//     PlcTask Inputs/GVL_iXlinker.EtherCAT_Master_EJxxxx.Beckhoff_EJ7xxx.A_0004_EJ7047_0000_0018.ENC_Status_compact.Status/Status_of_input_B <-> ENC Status compact/Status/Status of input B
//     PlcTask Inputs/GVL_iXlinker.EtherCAT_Master_EJxxxx.Beckhoff_EJ7xxx.A_0004_EJ7047_0000_0018.ENC_Status_compact.Status/Status_of_input_C <-> ENC Status compact/Status/Status of input C
//     PlcTask Inputs/GVL_iXlinker.EtherCAT_Master_EJxxxx.Beckhoff_EJ7xxx.A_0004_EJ7047_0000_0018.ENC_Status_compact.Status/Status_of_extern_latch <-> ENC Status compact/Status/Status of extern latch
//     PlcTask Inputs/GVL_iXlinker.EtherCAT_Master_EJxxxx.Beckhoff_EJ7xxx.A_0004_EJ7047_0000_0018.ENC_Status_compact.Status/Sync_error <-> ENC Status compact/Status/Sync error
//     PlcTask Inputs/GVL_iXlinker.EtherCAT_Master_EJxxxx.Beckhoff_EJ7xxx.A_0004_EJ7047_0000_0018.ENC_Status_compact.Status/TxPDO_Toggle <-> ENC Status compact/Status/TxPDO Toggle
//     PlcTask Inputs/GVL_iXlinker.EtherCAT_Master_EJxxxx.Beckhoff_EJ7xxx.A_0004_EJ7047_0000_0018.ENC_Status_compact.Counter_value <-> ENC Status compact/Counter value
//     PlcTask Inputs/GVL_iXlinker.EtherCAT_Master_EJxxxx.Beckhoff_EJ7xxx.A_0004_EJ7047_0000_0018.ENC_Status_compact.Latch_value <-> ENC Status compact/Latch value
//     PlcTask Inputs/GVL_iXlinker.EtherCAT_Master_EJxxxx.Beckhoff_EJ7xxx.A_0004_EJ7047_0000_0018.STM_Status.Status/Ready_to_enable <-> STM Status/Status/Ready to enable
//     PlcTask Inputs/GVL_iXlinker.EtherCAT_Master_EJxxxx.Beckhoff_EJ7xxx.A_0004_EJ7047_0000_0018.STM_Status.Status/Ready <-> STM Status/Status/Ready
//     PlcTask Inputs/GVL_iXlinker.EtherCAT_Master_EJxxxx.Beckhoff_EJ7xxx.A_0004_EJ7047_0000_0018.STM_Status.Status/Warning <-> STM Status/Status/Warning
//     PlcTask Inputs/GVL_iXlinker.EtherCAT_Master_EJxxxx.Beckhoff_EJ7xxx.A_0004_EJ7047_0000_0018.STM_Status.Status/Error <-> STM Status/Status/Error
//     PlcTask Inputs/GVL_iXlinker.EtherCAT_Master_EJxxxx.Beckhoff_EJ7xxx.A_0004_EJ7047_0000_0018.STM_Status.Status/Moving_positive <-> STM Status/Status/Moving positive
//     PlcTask Inputs/GVL_iXlinker.EtherCAT_Master_EJxxxx.Beckhoff_EJ7xxx.A_0004_EJ7047_0000_0018.STM_Status.Status/Moving_negative <-> STM Status/Status/Moving negative
//     PlcTask Inputs/GVL_iXlinker.EtherCAT_Master_EJxxxx.Beckhoff_EJ7xxx.A_0004_EJ7047_0000_0018.STM_Status.Status/Torque_reduced <-> STM Status/Status/Torque reduced
//     PlcTask Inputs/GVL_iXlinker.EtherCAT_Master_EJxxxx.Beckhoff_EJ7xxx.A_0004_EJ7047_0000_0018.STM_Status.Status/Motor_stall <-> STM Status/Status/Motor stall
//     PlcTask Inputs/GVL_iXlinker.EtherCAT_Master_EJxxxx.Beckhoff_EJ7xxx.A_0004_EJ7047_0000_0018.STM_Status.Status/Digital_input_1 <-> STM Status/Status/Digital input 1
//     PlcTask Inputs/GVL_iXlinker.EtherCAT_Master_EJxxxx.Beckhoff_EJ7xxx.A_0004_EJ7047_0000_0018.STM_Status.Status/Digital_input_2 <-> STM Status/Status/Digital input 2
//     PlcTask Inputs/GVL_iXlinker.EtherCAT_Master_EJxxxx.Beckhoff_EJ7xxx.A_0004_EJ7047_0000_0018.STM_Status.Status/Sync_error <-> STM Status/Status/Sync error
//     PlcTask Inputs/GVL_iXlinker.EtherCAT_Master_EJxxxx.Beckhoff_EJ7xxx.A_0004_EJ7047_0000_0018.STM_Status.Status/TxPDO_Toggle <-> STM Status/Status/TxPDO Toggle
//     PlcTask Outputs/GVL_iXlinker.EtherCAT_Master_EJxxxx.Beckhoff_EJ7xxx.A_0004_EJ7047_0000_0018.ENC_Control_compact.Control/Enable_latch_C <-> ENC Control compact/Control/Enable latch C
//     PlcTask Outputs/GVL_iXlinker.EtherCAT_Master_EJxxxx.Beckhoff_EJ7xxx.A_0004_EJ7047_0000_0018.ENC_Control_compact.Control/Enable_latch_extern_on_positive_edge <-> ENC Control compact/Control/Enable latch extern on positive edge
//     PlcTask Outputs/GVL_iXlinker.EtherCAT_Master_EJxxxx.Beckhoff_EJ7xxx.A_0004_EJ7047_0000_0018.ENC_Control_compact.Control/Set_counter <-> ENC Control compact/Control/Set counter
//     PlcTask Outputs/GVL_iXlinker.EtherCAT_Master_EJxxxx.Beckhoff_EJ7xxx.A_0004_EJ7047_0000_0018.ENC_Control_compact.Control/Enable_latch_extern_on_negative_edge <-> ENC Control compact/Control/Enable latch extern on negative edge
//     PlcTask Outputs/GVL_iXlinker.EtherCAT_Master_EJxxxx.Beckhoff_EJ7xxx.A_0004_EJ7047_0000_0018.ENC_Control_compact.Set_counter_value <-> ENC Control compact/Set counter value
//     PlcTask Outputs/GVL_iXlinker.EtherCAT_Master_EJxxxx.Beckhoff_EJ7xxx.A_0004_EJ7047_0000_0018.STM_Control.Control/Enable <-> STM Control/Control/Enable
//     PlcTask Outputs/GVL_iXlinker.EtherCAT_Master_EJxxxx.Beckhoff_EJ7xxx.A_0004_EJ7047_0000_0018.STM_Control.Control/Reset <-> STM Control/Control/Reset
//     PlcTask Outputs/GVL_iXlinker.EtherCAT_Master_EJxxxx.Beckhoff_EJ7xxx.A_0004_EJ7047_0000_0018.STM_Control.Control/Reduce_torque <-> STM Control/Control/Reduce torque
//     PlcTask Outputs/GVL_iXlinker.EtherCAT_Master_EJxxxx.Beckhoff_EJ7xxx.A_0004_EJ7047_0000_0018.STM_Control.Control/Digital_output_1 <-> STM Control/Control/Digital output 1
//     PlcTask Outputs/GVL_iXlinker.EtherCAT_Master_EJxxxx.Beckhoff_EJ7xxx.A_0004_EJ7047_0000_0018.STM_Velocity.Velocity <-> STM Velocity/Velocity
//     PlcTask Inputs/GVL_iXlinker.EtherCAT_Master_EJxxxx.Beckhoff_EJ7xxx.A_0004_EJ7047_0000_0018.WcState.WcState <-> WcState/WcState
//     PlcTask Inputs/GVL_iXlinker.EtherCAT_Master_EJxxxx.Beckhoff_EJ7xxx.A_0004_EJ7047_0000_0018.WcState.InputToggle <-> WcState/InputToggle
//     PlcTask Inputs/GVL_iXlinker.EtherCAT_Master_EJxxxx.Beckhoff_EJ7xxx.A_0004_EJ7047_0000_0018.InfoData.AdsAddr <-> InfoData/AdsAddr
//     PlcTask Inputs/GVL_iXlinker.EtherCAT_Master_EJxxxx.Beckhoff_EJ7xxx.A_0004_EJ7047_0000_0018.InfoData.Chn0 <-> InfoData/Chn0
//     PlcTask Inputs/GVL_iXlinker.EtherCAT_Master_EJxxxx.Beckhoff_EJ7xxx.A_0004_EJ7047_0000_0018.InfoData.Chn1 <-> InfoData/Chn1
//     PlcTask Inputs/GVL_iXlinker.EtherCAT_Master_EJxxxx.Beckhoff_EJ7xxx.A_0004_EJ7047_0000_0018.InfoData.State <-> InfoData/State
//   PLC/PLC Instance <-> EtherCAT Master EJxxxx/Beckhoff EJ7xxx/A_0005(EJ7047-0000-0019)
//     PlcTask Inputs/GVL_iXlinker.EtherCAT_Master_EJxxxx.Beckhoff_EJ7xxx.A_0005_EJ7047_0000_0019.ENC_Status_compact.Status/Latch_C_valid <-> ENC Status compact/Status/Latch C valid
//     PlcTask Inputs/GVL_iXlinker.EtherCAT_Master_EJxxxx.Beckhoff_EJ7xxx.A_0005_EJ7047_0000_0019.ENC_Status_compact.Status/Latch_extern_valid <-> ENC Status compact/Status/Latch extern valid
//     PlcTask Inputs/GVL_iXlinker.EtherCAT_Master_EJxxxx.Beckhoff_EJ7xxx.A_0005_EJ7047_0000_0019.ENC_Status_compact.Status/Set_counter_done <-> ENC Status compact/Status/Set counter done
//     PlcTask Inputs/GVL_iXlinker.EtherCAT_Master_EJxxxx.Beckhoff_EJ7xxx.A_0005_EJ7047_0000_0019.ENC_Status_compact.Status/Counter_underflow <-> ENC Status compact/Status/Counter underflow
//     PlcTask Inputs/GVL_iXlinker.EtherCAT_Master_EJxxxx.Beckhoff_EJ7xxx.A_0005_EJ7047_0000_0019.ENC_Status_compact.Status/Counter_overflow <-> ENC Status compact/Status/Counter overflow
//     PlcTask Inputs/GVL_iXlinker.EtherCAT_Master_EJxxxx.Beckhoff_EJ7xxx.A_0005_EJ7047_0000_0019.ENC_Status_compact.Status/Extrapolation_stall <-> ENC Status compact/Status/Extrapolation stall
//     PlcTask Inputs/GVL_iXlinker.EtherCAT_Master_EJxxxx.Beckhoff_EJ7xxx.A_0005_EJ7047_0000_0019.ENC_Status_compact.Status/Status_of_input_A <-> ENC Status compact/Status/Status of input A
//     PlcTask Inputs/GVL_iXlinker.EtherCAT_Master_EJxxxx.Beckhoff_EJ7xxx.A_0005_EJ7047_0000_0019.ENC_Status_compact.Status/Status_of_input_B <-> ENC Status compact/Status/Status of input B
//     PlcTask Inputs/GVL_iXlinker.EtherCAT_Master_EJxxxx.Beckhoff_EJ7xxx.A_0005_EJ7047_0000_0019.ENC_Status_compact.Status/Status_of_input_C <-> ENC Status compact/Status/Status of input C
//     PlcTask Inputs/GVL_iXlinker.EtherCAT_Master_EJxxxx.Beckhoff_EJ7xxx.A_0005_EJ7047_0000_0019.ENC_Status_compact.Status/Status_of_extern_latch <-> ENC Status compact/Status/Status of extern latch
//     PlcTask Inputs/GVL_iXlinker.EtherCAT_Master_EJxxxx.Beckhoff_EJ7xxx.A_0005_EJ7047_0000_0019.ENC_Status_compact.Status/Sync_error <-> ENC Status compact/Status/Sync error
//     PlcTask Inputs/GVL_iXlinker.EtherCAT_Master_EJxxxx.Beckhoff_EJ7xxx.A_0005_EJ7047_0000_0019.ENC_Status_compact.Status/TxPDO_Toggle <-> ENC Status compact/Status/TxPDO Toggle
//     PlcTask Inputs/GVL_iXlinker.EtherCAT_Master_EJxxxx.Beckhoff_EJ7xxx.A_0005_EJ7047_0000_0019.ENC_Status_compact.Counter_value <-> ENC Status compact/Counter value
//     PlcTask Inputs/GVL_iXlinker.EtherCAT_Master_EJxxxx.Beckhoff_EJ7xxx.A_0005_EJ7047_0000_0019.ENC_Status_compact.Latch_value <-> ENC Status compact/Latch value
//     PlcTask Inputs/GVL_iXlinker.EtherCAT_Master_EJxxxx.Beckhoff_EJ7xxx.A_0005_EJ7047_0000_0019.STM_Status.Status/Ready_to_enable <-> STM Status/Status/Ready to enable
//     PlcTask Inputs/GVL_iXlinker.EtherCAT_Master_EJxxxx.Beckhoff_EJ7xxx.A_0005_EJ7047_0000_0019.STM_Status.Status/Ready <-> STM Status/Status/Ready
//     PlcTask Inputs/GVL_iXlinker.EtherCAT_Master_EJxxxx.Beckhoff_EJ7xxx.A_0005_EJ7047_0000_0019.STM_Status.Status/Warning <-> STM Status/Status/Warning
//     PlcTask Inputs/GVL_iXlinker.EtherCAT_Master_EJxxxx.Beckhoff_EJ7xxx.A_0005_EJ7047_0000_0019.STM_Status.Status/Error <-> STM Status/Status/Error
//     PlcTask Inputs/GVL_iXlinker.EtherCAT_Master_EJxxxx.Beckhoff_EJ7xxx.A_0005_EJ7047_0000_0019.STM_Status.Status/Moving_positive <-> STM Status/Status/Moving positive
//     PlcTask Inputs/GVL_iXlinker.EtherCAT_Master_EJxxxx.Beckhoff_EJ7xxx.A_0005_EJ7047_0000_0019.STM_Status.Status/Moving_negative <-> STM Status/Status/Moving negative
//     PlcTask Inputs/GVL_iXlinker.EtherCAT_Master_EJxxxx.Beckhoff_EJ7xxx.A_0005_EJ7047_0000_0019.STM_Status.Status/Torque_reduced <-> STM Status/Status/Torque reduced
//     PlcTask Inputs/GVL_iXlinker.EtherCAT_Master_EJxxxx.Beckhoff_EJ7xxx.A_0005_EJ7047_0000_0019.STM_Status.Status/Motor_stall <-> STM Status/Status/Motor stall
//     PlcTask Inputs/GVL_iXlinker.EtherCAT_Master_EJxxxx.Beckhoff_EJ7xxx.A_0005_EJ7047_0000_0019.STM_Status.Status/Digital_input_1 <-> STM Status/Status/Digital input 1
//     PlcTask Inputs/GVL_iXlinker.EtherCAT_Master_EJxxxx.Beckhoff_EJ7xxx.A_0005_EJ7047_0000_0019.STM_Status.Status/Digital_input_2 <-> STM Status/Status/Digital input 2
//     PlcTask Inputs/GVL_iXlinker.EtherCAT_Master_EJxxxx.Beckhoff_EJ7xxx.A_0005_EJ7047_0000_0019.STM_Status.Status/Sync_error <-> STM Status/Status/Sync error
//     PlcTask Inputs/GVL_iXlinker.EtherCAT_Master_EJxxxx.Beckhoff_EJ7xxx.A_0005_EJ7047_0000_0019.STM_Status.Status/TxPDO_Toggle <-> STM Status/Status/TxPDO Toggle
//     PlcTask Outputs/GVL_iXlinker.EtherCAT_Master_EJxxxx.Beckhoff_EJ7xxx.A_0005_EJ7047_0000_0019.ENC_Control_compact.Control/Enable_latch_C <-> ENC Control compact/Control/Enable latch C
//     PlcTask Outputs/GVL_iXlinker.EtherCAT_Master_EJxxxx.Beckhoff_EJ7xxx.A_0005_EJ7047_0000_0019.ENC_Control_compact.Control/Enable_latch_extern_on_positive_edge <-> ENC Control compact/Control/Enable latch extern on positive edge
//     PlcTask Outputs/GVL_iXlinker.EtherCAT_Master_EJxxxx.Beckhoff_EJ7xxx.A_0005_EJ7047_0000_0019.ENC_Control_compact.Control/Set_counter <-> ENC Control compact/Control/Set counter
//     PlcTask Outputs/GVL_iXlinker.EtherCAT_Master_EJxxxx.Beckhoff_EJ7xxx.A_0005_EJ7047_0000_0019.ENC_Control_compact.Control/Enable_latch_extern_on_negative_edge <-> ENC Control compact/Control/Enable latch extern on negative edge
//     PlcTask Outputs/GVL_iXlinker.EtherCAT_Master_EJxxxx.Beckhoff_EJ7xxx.A_0005_EJ7047_0000_0019.ENC_Control_compact.Set_counter_value <-> ENC Control compact/Set counter value
//     PlcTask Outputs/GVL_iXlinker.EtherCAT_Master_EJxxxx.Beckhoff_EJ7xxx.A_0005_EJ7047_0000_0019.STM_Control.Control/Enable <-> STM Control/Control/Enable
//     PlcTask Outputs/GVL_iXlinker.EtherCAT_Master_EJxxxx.Beckhoff_EJ7xxx.A_0005_EJ7047_0000_0019.STM_Control.Control/Reset <-> STM Control/Control/Reset
//     PlcTask Outputs/GVL_iXlinker.EtherCAT_Master_EJxxxx.Beckhoff_EJ7xxx.A_0005_EJ7047_0000_0019.STM_Control.Control/Reduce_torque <-> STM Control/Control/Reduce torque
//     PlcTask Outputs/GVL_iXlinker.EtherCAT_Master_EJxxxx.Beckhoff_EJ7xxx.A_0005_EJ7047_0000_0019.STM_Control.Control/Digital_output_1 <-> STM Control/Control/Digital output 1
//     PlcTask Outputs/GVL_iXlinker.EtherCAT_Master_EJxxxx.Beckhoff_EJ7xxx.A_0005_EJ7047_0000_0019.STM_Velocity.Velocity <-> STM Velocity/Velocity
//     PlcTask Inputs/GVL_iXlinker.EtherCAT_Master_EJxxxx.Beckhoff_EJ7xxx.A_0005_EJ7047_0000_0019.WcState.WcState <-> WcState/WcState
//     PlcTask Inputs/GVL_iXlinker.EtherCAT_Master_EJxxxx.Beckhoff_EJ7xxx.A_0005_EJ7047_0000_0019.WcState.InputToggle <-> WcState/InputToggle
//     PlcTask Inputs/GVL_iXlinker.EtherCAT_Master_EJxxxx.Beckhoff_EJ7xxx.A_0005_EJ7047_0000_0019.InfoData.AdsAddr <-> InfoData/AdsAddr
//     PlcTask Inputs/GVL_iXlinker.EtherCAT_Master_EJxxxx.Beckhoff_EJ7xxx.A_0005_EJ7047_0000_0019.InfoData.Chn0 <-> InfoData/Chn0
//     PlcTask Inputs/GVL_iXlinker.EtherCAT_Master_EJxxxx.Beckhoff_EJ7xxx.A_0005_EJ7047_0000_0019.InfoData.Chn1 <-> InfoData/Chn1
//     PlcTask Inputs/GVL_iXlinker.EtherCAT_Master_EJxxxx.Beckhoff_EJ7xxx.A_0005_EJ7047_0000_0019.InfoData.State <-> InfoData/State
//   PLC/PLC Instance <-> EtherCAT Master EJxxxx/Beckhoff EJ7xxx/A_0006(EJ7047-0000-0020)
//     PlcTask Inputs/GVL_iXlinker.EtherCAT_Master_EJxxxx.Beckhoff_EJ7xxx.A_0006_EJ7047_0000_0020.ENC_Status_compact.Status/Latch_C_valid <-> ENC Status compact/Status/Latch C valid
//     PlcTask Inputs/GVL_iXlinker.EtherCAT_Master_EJxxxx.Beckhoff_EJ7xxx.A_0006_EJ7047_0000_0020.ENC_Status_compact.Status/Latch_extern_valid <-> ENC Status compact/Status/Latch extern valid
//     PlcTask Inputs/GVL_iXlinker.EtherCAT_Master_EJxxxx.Beckhoff_EJ7xxx.A_0006_EJ7047_0000_0020.ENC_Status_compact.Status/Set_counter_done <-> ENC Status compact/Status/Set counter done
//     PlcTask Inputs/GVL_iXlinker.EtherCAT_Master_EJxxxx.Beckhoff_EJ7xxx.A_0006_EJ7047_0000_0020.ENC_Status_compact.Status/Counter_underflow <-> ENC Status compact/Status/Counter underflow
//     PlcTask Inputs/GVL_iXlinker.EtherCAT_Master_EJxxxx.Beckhoff_EJ7xxx.A_0006_EJ7047_0000_0020.ENC_Status_compact.Status/Counter_overflow <-> ENC Status compact/Status/Counter overflow
//     PlcTask Inputs/GVL_iXlinker.EtherCAT_Master_EJxxxx.Beckhoff_EJ7xxx.A_0006_EJ7047_0000_0020.ENC_Status_compact.Status/Extrapolation_stall <-> ENC Status compact/Status/Extrapolation stall
//     PlcTask Inputs/GVL_iXlinker.EtherCAT_Master_EJxxxx.Beckhoff_EJ7xxx.A_0006_EJ7047_0000_0020.ENC_Status_compact.Status/Status_of_input_A <-> ENC Status compact/Status/Status of input A
//     PlcTask Inputs/GVL_iXlinker.EtherCAT_Master_EJxxxx.Beckhoff_EJ7xxx.A_0006_EJ7047_0000_0020.ENC_Status_compact.Status/Status_of_input_B <-> ENC Status compact/Status/Status of input B
//     PlcTask Inputs/GVL_iXlinker.EtherCAT_Master_EJxxxx.Beckhoff_EJ7xxx.A_0006_EJ7047_0000_0020.ENC_Status_compact.Status/Status_of_input_C <-> ENC Status compact/Status/Status of input C
//     PlcTask Inputs/GVL_iXlinker.EtherCAT_Master_EJxxxx.Beckhoff_EJ7xxx.A_0006_EJ7047_0000_0020.ENC_Status_compact.Status/Status_of_extern_latch <-> ENC Status compact/Status/Status of extern latch
//     PlcTask Inputs/GVL_iXlinker.EtherCAT_Master_EJxxxx.Beckhoff_EJ7xxx.A_0006_EJ7047_0000_0020.ENC_Status_compact.Status/Sync_error <-> ENC Status compact/Status/Sync error
//     PlcTask Inputs/GVL_iXlinker.EtherCAT_Master_EJxxxx.Beckhoff_EJ7xxx.A_0006_EJ7047_0000_0020.ENC_Status_compact.Status/TxPDO_Toggle <-> ENC Status compact/Status/TxPDO Toggle
//     PlcTask Inputs/GVL_iXlinker.EtherCAT_Master_EJxxxx.Beckhoff_EJ7xxx.A_0006_EJ7047_0000_0020.ENC_Status_compact.Counter_value <-> ENC Status compact/Counter value
//     PlcTask Inputs/GVL_iXlinker.EtherCAT_Master_EJxxxx.Beckhoff_EJ7xxx.A_0006_EJ7047_0000_0020.ENC_Status_compact.Latch_value <-> ENC Status compact/Latch value
//     PlcTask Inputs/GVL_iXlinker.EtherCAT_Master_EJxxxx.Beckhoff_EJ7xxx.A_0006_EJ7047_0000_0020.STM_Status.Status/Ready_to_enable <-> STM Status/Status/Ready to enable
//     PlcTask Inputs/GVL_iXlinker.EtherCAT_Master_EJxxxx.Beckhoff_EJ7xxx.A_0006_EJ7047_0000_0020.STM_Status.Status/Ready <-> STM Status/Status/Ready
//     PlcTask Inputs/GVL_iXlinker.EtherCAT_Master_EJxxxx.Beckhoff_EJ7xxx.A_0006_EJ7047_0000_0020.STM_Status.Status/Warning <-> STM Status/Status/Warning
//     PlcTask Inputs/GVL_iXlinker.EtherCAT_Master_EJxxxx.Beckhoff_EJ7xxx.A_0006_EJ7047_0000_0020.STM_Status.Status/Error <-> STM Status/Status/Error
//     PlcTask Inputs/GVL_iXlinker.EtherCAT_Master_EJxxxx.Beckhoff_EJ7xxx.A_0006_EJ7047_0000_0020.STM_Status.Status/Moving_positive <-> STM Status/Status/Moving positive
//     PlcTask Inputs/GVL_iXlinker.EtherCAT_Master_EJxxxx.Beckhoff_EJ7xxx.A_0006_EJ7047_0000_0020.STM_Status.Status/Moving_negative <-> STM Status/Status/Moving negative
//     PlcTask Inputs/GVL_iXlinker.EtherCAT_Master_EJxxxx.Beckhoff_EJ7xxx.A_0006_EJ7047_0000_0020.STM_Status.Status/Torque_reduced <-> STM Status/Status/Torque reduced
//     PlcTask Inputs/GVL_iXlinker.EtherCAT_Master_EJxxxx.Beckhoff_EJ7xxx.A_0006_EJ7047_0000_0020.STM_Status.Status/Motor_stall <-> STM Status/Status/Motor stall
//     PlcTask Inputs/GVL_iXlinker.EtherCAT_Master_EJxxxx.Beckhoff_EJ7xxx.A_0006_EJ7047_0000_0020.STM_Status.Status/Digital_input_1 <-> STM Status/Status/Digital input 1
//     PlcTask Inputs/GVL_iXlinker.EtherCAT_Master_EJxxxx.Beckhoff_EJ7xxx.A_0006_EJ7047_0000_0020.STM_Status.Status/Digital_input_2 <-> STM Status/Status/Digital input 2
//     PlcTask Inputs/GVL_iXlinker.EtherCAT_Master_EJxxxx.Beckhoff_EJ7xxx.A_0006_EJ7047_0000_0020.STM_Status.Status/Sync_error <-> STM Status/Status/Sync error
//     PlcTask Inputs/GVL_iXlinker.EtherCAT_Master_EJxxxx.Beckhoff_EJ7xxx.A_0006_EJ7047_0000_0020.STM_Status.Status/TxPDO_Toggle <-> STM Status/Status/TxPDO Toggle
//     PlcTask Outputs/GVL_iXlinker.EtherCAT_Master_EJxxxx.Beckhoff_EJ7xxx.A_0006_EJ7047_0000_0020.ENC_Control_compact.Control/Enable_latch_C <-> ENC Control compact/Control/Enable latch C
//     PlcTask Outputs/GVL_iXlinker.EtherCAT_Master_EJxxxx.Beckhoff_EJ7xxx.A_0006_EJ7047_0000_0020.ENC_Control_compact.Control/Enable_latch_extern_on_positive_edge <-> ENC Control compact/Control/Enable latch extern on positive edge
//     PlcTask Outputs/GVL_iXlinker.EtherCAT_Master_EJxxxx.Beckhoff_EJ7xxx.A_0006_EJ7047_0000_0020.ENC_Control_compact.Control/Set_counter <-> ENC Control compact/Control/Set counter
//     PlcTask Outputs/GVL_iXlinker.EtherCAT_Master_EJxxxx.Beckhoff_EJ7xxx.A_0006_EJ7047_0000_0020.ENC_Control_compact.Control/Enable_latch_extern_on_negative_edge <-> ENC Control compact/Control/Enable latch extern on negative edge
//     PlcTask Outputs/GVL_iXlinker.EtherCAT_Master_EJxxxx.Beckhoff_EJ7xxx.A_0006_EJ7047_0000_0020.ENC_Control_compact.Set_counter_value <-> ENC Control compact/Set counter value
//     PlcTask Outputs/GVL_iXlinker.EtherCAT_Master_EJxxxx.Beckhoff_EJ7xxx.A_0006_EJ7047_0000_0020.STM_Control.Control/Enable <-> STM Control/Control/Enable
//     PlcTask Outputs/GVL_iXlinker.EtherCAT_Master_EJxxxx.Beckhoff_EJ7xxx.A_0006_EJ7047_0000_0020.STM_Control.Control/Reset <-> STM Control/Control/Reset
//     PlcTask Outputs/GVL_iXlinker.EtherCAT_Master_EJxxxx.Beckhoff_EJ7xxx.A_0006_EJ7047_0000_0020.STM_Control.Control/Reduce_torque <-> STM Control/Control/Reduce torque
//     PlcTask Outputs/GVL_iXlinker.EtherCAT_Master_EJxxxx.Beckhoff_EJ7xxx.A_0006_EJ7047_0000_0020.STM_Control.Control/Digital_output_1 <-> STM Control/Control/Digital output 1
//     PlcTask Outputs/GVL_iXlinker.EtherCAT_Master_EJxxxx.Beckhoff_EJ7xxx.A_0006_EJ7047_0000_0020.STM_Velocity.Velocity <-> STM Velocity/Velocity
//     PlcTask Inputs/GVL_iXlinker.EtherCAT_Master_EJxxxx.Beckhoff_EJ7xxx.A_0006_EJ7047_0000_0020.WcState.WcState <-> WcState/WcState
//     PlcTask Inputs/GVL_iXlinker.EtherCAT_Master_EJxxxx.Beckhoff_EJ7xxx.A_0006_EJ7047_0000_0020.WcState.InputToggle <-> WcState/InputToggle
//     PlcTask Inputs/GVL_iXlinker.EtherCAT_Master_EJxxxx.Beckhoff_EJ7xxx.A_0006_EJ7047_0000_0020.InfoData.AdsAddr <-> InfoData/AdsAddr
//     PlcTask Inputs/GVL_iXlinker.EtherCAT_Master_EJxxxx.Beckhoff_EJ7xxx.A_0006_EJ7047_0000_0020.InfoData.Chn0 <-> InfoData/Chn0
//     PlcTask Inputs/GVL_iXlinker.EtherCAT_Master_EJxxxx.Beckhoff_EJ7xxx.A_0006_EJ7047_0000_0020.InfoData.Chn1 <-> InfoData/Chn1
//     PlcTask Inputs/GVL_iXlinker.EtherCAT_Master_EJxxxx.Beckhoff_EJ7xxx.A_0006_EJ7047_0000_0020.InfoData.State <-> InfoData/State
//   PLC/PLC Instance <-> EtherCAT Master EJxxxx/Beckhoff EJ7xxx/A_0007(EJ7342-0000-0019)
//     PlcTask Inputs/GVL_iXlinker.EtherCAT_Master_EJxxxx.Beckhoff_EJ7xxx.A_0007_EJ7342_0000_0019.ENC_Status_compact_Channel_1.Status/Latch_extern_valid <-> ENC Status compact Channel 1/Status/Latch extern valid
//     PlcTask Inputs/GVL_iXlinker.EtherCAT_Master_EJxxxx.Beckhoff_EJ7xxx.A_0007_EJ7342_0000_0019.ENC_Status_compact_Channel_2.Status/Latch_extern_valid <-> ENC Status compact Channel 2/Status/Latch extern valid
//     PlcTask Inputs/GVL_iXlinker.EtherCAT_Master_EJxxxx.Beckhoff_EJ7xxx.A_0007_EJ7342_0000_0019.ENC_Status_compact_Channel_1.Status/Set_counter_done <-> ENC Status compact Channel 1/Status/Set counter done
//     PlcTask Inputs/GVL_iXlinker.EtherCAT_Master_EJxxxx.Beckhoff_EJ7xxx.A_0007_EJ7342_0000_0019.ENC_Status_compact_Channel_2.Status/Set_counter_done <-> ENC Status compact Channel 2/Status/Set counter done
//     PlcTask Inputs/GVL_iXlinker.EtherCAT_Master_EJxxxx.Beckhoff_EJ7xxx.A_0007_EJ7342_0000_0019.ENC_Status_compact_Channel_1.Status/Counter_underflow <-> ENC Status compact Channel 1/Status/Counter underflow
//     PlcTask Inputs/GVL_iXlinker.EtherCAT_Master_EJxxxx.Beckhoff_EJ7xxx.A_0007_EJ7342_0000_0019.ENC_Status_compact_Channel_2.Status/Counter_underflow <-> ENC Status compact Channel 2/Status/Counter underflow
//     PlcTask Inputs/GVL_iXlinker.EtherCAT_Master_EJxxxx.Beckhoff_EJ7xxx.A_0007_EJ7342_0000_0019.ENC_Status_compact_Channel_1.Status/Counter_overflow <-> ENC Status compact Channel 1/Status/Counter overflow
//     PlcTask Inputs/GVL_iXlinker.EtherCAT_Master_EJxxxx.Beckhoff_EJ7xxx.A_0007_EJ7342_0000_0019.ENC_Status_compact_Channel_2.Status/Counter_overflow <-> ENC Status compact Channel 2/Status/Counter overflow
//     PlcTask Inputs/GVL_iXlinker.EtherCAT_Master_EJxxxx.Beckhoff_EJ7xxx.A_0007_EJ7342_0000_0019.ENC_Status_compact_Channel_1.Status/Extrapolation_stall <-> ENC Status compact Channel 1/Status/Extrapolation stall
//     PlcTask Inputs/GVL_iXlinker.EtherCAT_Master_EJxxxx.Beckhoff_EJ7xxx.A_0007_EJ7342_0000_0019.ENC_Status_compact_Channel_2.Status/Extrapolation_stall <-> ENC Status compact Channel 2/Status/Extrapolation stall
//     PlcTask Inputs/GVL_iXlinker.EtherCAT_Master_EJxxxx.Beckhoff_EJ7xxx.A_0007_EJ7342_0000_0019.ENC_Status_compact_Channel_1.Status/Status_of_input_A <-> ENC Status compact Channel 1/Status/Status of input A
//     PlcTask Inputs/GVL_iXlinker.EtherCAT_Master_EJxxxx.Beckhoff_EJ7xxx.A_0007_EJ7342_0000_0019.ENC_Status_compact_Channel_2.Status/Status_of_input_A <-> ENC Status compact Channel 2/Status/Status of input A
//     PlcTask Inputs/GVL_iXlinker.EtherCAT_Master_EJxxxx.Beckhoff_EJ7xxx.A_0007_EJ7342_0000_0019.ENC_Status_compact_Channel_1.Status/Status_of_input_B <-> ENC Status compact Channel 1/Status/Status of input B
//     PlcTask Inputs/GVL_iXlinker.EtherCAT_Master_EJxxxx.Beckhoff_EJ7xxx.A_0007_EJ7342_0000_0019.ENC_Status_compact_Channel_2.Status/Status_of_input_B <-> ENC Status compact Channel 2/Status/Status of input B
//     PlcTask Inputs/GVL_iXlinker.EtherCAT_Master_EJxxxx.Beckhoff_EJ7xxx.A_0007_EJ7342_0000_0019.ENC_Status_compact_Channel_1.Status/Status_of_extern_latch <-> ENC Status compact Channel 1/Status/Status of extern latch
//     PlcTask Inputs/GVL_iXlinker.EtherCAT_Master_EJxxxx.Beckhoff_EJ7xxx.A_0007_EJ7342_0000_0019.ENC_Status_compact_Channel_2.Status/Status_of_extern_latch <-> ENC Status compact Channel 2/Status/Status of extern latch
//     PlcTask Inputs/GVL_iXlinker.EtherCAT_Master_EJxxxx.Beckhoff_EJ7xxx.A_0007_EJ7342_0000_0019.ENC_Status_compact_Channel_1.Status/Sync_error <-> ENC Status compact Channel 1/Status/Sync error
//     PlcTask Inputs/GVL_iXlinker.EtherCAT_Master_EJxxxx.Beckhoff_EJ7xxx.A_0007_EJ7342_0000_0019.ENC_Status_compact_Channel_2.Status/Sync_error <-> ENC Status compact Channel 2/Status/Sync error
//     PlcTask Inputs/GVL_iXlinker.EtherCAT_Master_EJxxxx.Beckhoff_EJ7xxx.A_0007_EJ7342_0000_0019.ENC_Status_compact_Channel_1.Status/TxPDO_Toggle <-> ENC Status compact Channel 1/Status/TxPDO Toggle
//     PlcTask Inputs/GVL_iXlinker.EtherCAT_Master_EJxxxx.Beckhoff_EJ7xxx.A_0007_EJ7342_0000_0019.ENC_Status_compact_Channel_2.Status/TxPDO_Toggle <-> ENC Status compact Channel 2/Status/TxPDO Toggle
//     PlcTask Inputs/GVL_iXlinker.EtherCAT_Master_EJxxxx.Beckhoff_EJ7xxx.A_0007_EJ7342_0000_0019.ENC_Status_compact_Channel_1.Counter_value <-> ENC Status compact Channel 1/Counter value
//     PlcTask Inputs/GVL_iXlinker.EtherCAT_Master_EJxxxx.Beckhoff_EJ7xxx.A_0007_EJ7342_0000_0019.ENC_Status_compact_Channel_2.Counter_value <-> ENC Status compact Channel 2/Counter value
//     PlcTask Inputs/GVL_iXlinker.EtherCAT_Master_EJxxxx.Beckhoff_EJ7xxx.A_0007_EJ7342_0000_0019.ENC_Status_compact_Channel_1.Latch_value <-> ENC Status compact Channel 1/Latch value
//     PlcTask Inputs/GVL_iXlinker.EtherCAT_Master_EJxxxx.Beckhoff_EJ7xxx.A_0007_EJ7342_0000_0019.ENC_Status_compact_Channel_2.Latch_value <-> ENC Status compact Channel 2/Latch value
//     PlcTask Inputs/GVL_iXlinker.EtherCAT_Master_EJxxxx.Beckhoff_EJ7xxx.A_0007_EJ7342_0000_0019.DCM_Status_Channel_1.Status/Ready_to_enable <-> DCM Status Channel 1/Status/Ready to enable
//     PlcTask Inputs/GVL_iXlinker.EtherCAT_Master_EJxxxx.Beckhoff_EJ7xxx.A_0007_EJ7342_0000_0019.DCM_Status_Channel_2.Status/Ready_to_enable <-> DCM Status Channel 2/Status/Ready to enable
//     PlcTask Inputs/GVL_iXlinker.EtherCAT_Master_EJxxxx.Beckhoff_EJ7xxx.A_0007_EJ7342_0000_0019.DCM_Status_Channel_1.Status/Ready <-> DCM Status Channel 1/Status/Ready
//     PlcTask Inputs/GVL_iXlinker.EtherCAT_Master_EJxxxx.Beckhoff_EJ7xxx.A_0007_EJ7342_0000_0019.DCM_Status_Channel_2.Status/Ready <-> DCM Status Channel 2/Status/Ready
//     PlcTask Inputs/GVL_iXlinker.EtherCAT_Master_EJxxxx.Beckhoff_EJ7xxx.A_0007_EJ7342_0000_0019.DCM_Status_Channel_1.Status/Warning <-> DCM Status Channel 1/Status/Warning
//     PlcTask Inputs/GVL_iXlinker.EtherCAT_Master_EJxxxx.Beckhoff_EJ7xxx.A_0007_EJ7342_0000_0019.DCM_Status_Channel_2.Status/Warning <-> DCM Status Channel 2/Status/Warning
//     PlcTask Inputs/GVL_iXlinker.EtherCAT_Master_EJxxxx.Beckhoff_EJ7xxx.A_0007_EJ7342_0000_0019.DCM_Status_Channel_1.Status/Error <-> DCM Status Channel 1/Status/Error
//     PlcTask Inputs/GVL_iXlinker.EtherCAT_Master_EJxxxx.Beckhoff_EJ7xxx.A_0007_EJ7342_0000_0019.DCM_Status_Channel_2.Status/Error <-> DCM Status Channel 2/Status/Error
//     PlcTask Inputs/GVL_iXlinker.EtherCAT_Master_EJxxxx.Beckhoff_EJ7xxx.A_0007_EJ7342_0000_0019.DCM_Status_Channel_1.Status/Moving_positive <-> DCM Status Channel 1/Status/Moving positive
//     PlcTask Inputs/GVL_iXlinker.EtherCAT_Master_EJxxxx.Beckhoff_EJ7xxx.A_0007_EJ7342_0000_0019.DCM_Status_Channel_2.Status/Moving_positive <-> DCM Status Channel 2/Status/Moving positive
//     PlcTask Inputs/GVL_iXlinker.EtherCAT_Master_EJxxxx.Beckhoff_EJ7xxx.A_0007_EJ7342_0000_0019.DCM_Status_Channel_1.Status/Moving_negative <-> DCM Status Channel 1/Status/Moving negative
//     PlcTask Inputs/GVL_iXlinker.EtherCAT_Master_EJxxxx.Beckhoff_EJ7xxx.A_0007_EJ7342_0000_0019.DCM_Status_Channel_2.Status/Moving_negative <-> DCM Status Channel 2/Status/Moving negative
//     PlcTask Inputs/GVL_iXlinker.EtherCAT_Master_EJxxxx.Beckhoff_EJ7xxx.A_0007_EJ7342_0000_0019.DCM_Status_Channel_1.Status/Torque_reduced <-> DCM Status Channel 1/Status/Torque reduced
//     PlcTask Inputs/GVL_iXlinker.EtherCAT_Master_EJxxxx.Beckhoff_EJ7xxx.A_0007_EJ7342_0000_0019.DCM_Status_Channel_2.Status/Torque_reduced <-> DCM Status Channel 2/Status/Torque reduced
//     PlcTask Inputs/GVL_iXlinker.EtherCAT_Master_EJxxxx.Beckhoff_EJ7xxx.A_0007_EJ7342_0000_0019.DCM_Status_Channel_1.Status/Digital_input_1 <-> DCM Status Channel 1/Status/Digital input 1
//     PlcTask Inputs/GVL_iXlinker.EtherCAT_Master_EJxxxx.Beckhoff_EJ7xxx.A_0007_EJ7342_0000_0019.DCM_Status_Channel_1.Status/Digital_input_2 <-> DCM Status Channel 1/Status/Digital input 2
//     PlcTask Inputs/GVL_iXlinker.EtherCAT_Master_EJxxxx.Beckhoff_EJ7xxx.A_0007_EJ7342_0000_0019.DCM_Status_Channel_2.Status/Digital_input_1 <-> DCM Status Channel 2/Status/Digital input 1
//     PlcTask Inputs/GVL_iXlinker.EtherCAT_Master_EJxxxx.Beckhoff_EJ7xxx.A_0007_EJ7342_0000_0019.DCM_Status_Channel_2.Status/Digital_input_2 <-> DCM Status Channel 2/Status/Digital input 2
//     PlcTask Inputs/GVL_iXlinker.EtherCAT_Master_EJxxxx.Beckhoff_EJ7xxx.A_0007_EJ7342_0000_0019.DCM_Status_Channel_1.Status/Sync_error <-> DCM Status Channel 1/Status/Sync error
//     PlcTask Inputs/GVL_iXlinker.EtherCAT_Master_EJxxxx.Beckhoff_EJ7xxx.A_0007_EJ7342_0000_0019.DCM_Status_Channel_2.Status/Sync_error <-> DCM Status Channel 2/Status/Sync error
//     PlcTask Inputs/GVL_iXlinker.EtherCAT_Master_EJxxxx.Beckhoff_EJ7xxx.A_0007_EJ7342_0000_0019.DCM_Status_Channel_1.Status/TxPDO_Toggle <-> DCM Status Channel 1/Status/TxPDO Toggle
//     PlcTask Inputs/GVL_iXlinker.EtherCAT_Master_EJxxxx.Beckhoff_EJ7xxx.A_0007_EJ7342_0000_0019.DCM_Status_Channel_2.Status/TxPDO_Toggle <-> DCM Status Channel 2/Status/TxPDO Toggle
//     PlcTask Outputs/GVL_iXlinker.EtherCAT_Master_EJxxxx.Beckhoff_EJ7xxx.A_0007_EJ7342_0000_0019.ENC_Control_compact_Channel_1.Control/Enable_latch_extern_on_positive_edge <-> ENC Control compact Channel 1/Control/Enable latch extern on positive edge
//     PlcTask Outputs/GVL_iXlinker.EtherCAT_Master_EJxxxx.Beckhoff_EJ7xxx.A_0007_EJ7342_0000_0019.ENC_Control_compact_Channel_2.Control/Enable_latch_extern_on_positive_edge <-> ENC Control compact Channel 2/Control/Enable latch extern on positive edge
//     PlcTask Outputs/GVL_iXlinker.EtherCAT_Master_EJxxxx.Beckhoff_EJ7xxx.A_0007_EJ7342_0000_0019.ENC_Control_compact_Channel_1.Control/Set_counter <-> ENC Control compact Channel 1/Control/Set counter
//     PlcTask Outputs/GVL_iXlinker.EtherCAT_Master_EJxxxx.Beckhoff_EJ7xxx.A_0007_EJ7342_0000_0019.ENC_Control_compact_Channel_2.Control/Set_counter <-> ENC Control compact Channel 2/Control/Set counter
//     PlcTask Outputs/GVL_iXlinker.EtherCAT_Master_EJxxxx.Beckhoff_EJ7xxx.A_0007_EJ7342_0000_0019.ENC_Control_compact_Channel_1.Control/Enable_latch_extern_on_negative_edge <-> ENC Control compact Channel 1/Control/Enable latch extern on negative edge
//     PlcTask Outputs/GVL_iXlinker.EtherCAT_Master_EJxxxx.Beckhoff_EJ7xxx.A_0007_EJ7342_0000_0019.ENC_Control_compact_Channel_2.Control/Enable_latch_extern_on_negative_edge <-> ENC Control compact Channel 2/Control/Enable latch extern on negative edge
//     PlcTask Outputs/GVL_iXlinker.EtherCAT_Master_EJxxxx.Beckhoff_EJ7xxx.A_0007_EJ7342_0000_0019.ENC_Control_compact_Channel_1.Set_counter_value <-> ENC Control compact Channel 1/Set counter value
//     PlcTask Outputs/GVL_iXlinker.EtherCAT_Master_EJxxxx.Beckhoff_EJ7xxx.A_0007_EJ7342_0000_0019.ENC_Control_compact_Channel_2.Set_counter_value <-> ENC Control compact Channel 2/Set counter value
//     PlcTask Outputs/GVL_iXlinker.EtherCAT_Master_EJxxxx.Beckhoff_EJ7xxx.A_0007_EJ7342_0000_0019.DCM_Control_Channel_1.Control/Enable <-> DCM Control Channel 1/Control/Enable
//     PlcTask Outputs/GVL_iXlinker.EtherCAT_Master_EJxxxx.Beckhoff_EJ7xxx.A_0007_EJ7342_0000_0019.DCM_Control_Channel_2.Control/Enable <-> DCM Control Channel 2/Control/Enable
//     PlcTask Outputs/GVL_iXlinker.EtherCAT_Master_EJxxxx.Beckhoff_EJ7xxx.A_0007_EJ7342_0000_0019.DCM_Control_Channel_1.Control/Reset <-> DCM Control Channel 1/Control/Reset
//     PlcTask Outputs/GVL_iXlinker.EtherCAT_Master_EJxxxx.Beckhoff_EJ7xxx.A_0007_EJ7342_0000_0019.DCM_Control_Channel_2.Control/Reset <-> DCM Control Channel 2/Control/Reset
//     PlcTask Outputs/GVL_iXlinker.EtherCAT_Master_EJxxxx.Beckhoff_EJ7xxx.A_0007_EJ7342_0000_0019.DCM_Control_Channel_1.Control/Reduce_torque <-> DCM Control Channel 1/Control/Reduce torque
//     PlcTask Outputs/GVL_iXlinker.EtherCAT_Master_EJxxxx.Beckhoff_EJ7xxx.A_0007_EJ7342_0000_0019.DCM_Control_Channel_2.Control/Reduce_torque <-> DCM Control Channel 2/Control/Reduce torque
//     PlcTask Outputs/GVL_iXlinker.EtherCAT_Master_EJxxxx.Beckhoff_EJ7xxx.A_0007_EJ7342_0000_0019.DCM_Velocity_Channel_1.Velocity <-> DCM Velocity Channel 1/Velocity
//     PlcTask Outputs/GVL_iXlinker.EtherCAT_Master_EJxxxx.Beckhoff_EJ7xxx.A_0007_EJ7342_0000_0019.DCM_Velocity_Channel_2.Velocity <-> DCM Velocity Channel 2/Velocity
//     PlcTask Inputs/GVL_iXlinker.EtherCAT_Master_EJxxxx.Beckhoff_EJ7xxx.A_0007_EJ7342_0000_0019.WcState.WcState <-> WcState/WcState
//     PlcTask Inputs/GVL_iXlinker.EtherCAT_Master_EJxxxx.Beckhoff_EJ7xxx.A_0007_EJ7342_0000_0019.WcState.InputToggle <-> WcState/InputToggle
//     PlcTask Inputs/GVL_iXlinker.EtherCAT_Master_EJxxxx.Beckhoff_EJ7xxx.A_0007_EJ7342_0000_0019.InfoData.AdsAddr <-> InfoData/AdsAddr
//     PlcTask Inputs/GVL_iXlinker.EtherCAT_Master_EJxxxx.Beckhoff_EJ7xxx.A_0007_EJ7342_0000_0019.InfoData.Chn0 <-> InfoData/Chn0
//     PlcTask Inputs/GVL_iXlinker.EtherCAT_Master_EJxxxx.Beckhoff_EJ7xxx.A_0007_EJ7342_0000_0019.InfoData.Chn1 <-> InfoData/Chn1
//     PlcTask Inputs/GVL_iXlinker.EtherCAT_Master_EJxxxx.Beckhoff_EJ7xxx.A_0007_EJ7342_0000_0019.InfoData.Chn2 <-> InfoData/Chn2
//     PlcTask Inputs/GVL_iXlinker.EtherCAT_Master_EJxxxx.Beckhoff_EJ7xxx.A_0007_EJ7342_0000_0019.InfoData.Chn3 <-> InfoData/Chn3
//     PlcTask Inputs/GVL_iXlinker.EtherCAT_Master_EJxxxx.Beckhoff_EJ7xxx.A_0007_EJ7342_0000_0019.InfoData.State <-> InfoData/State
//   PLC/PLC Instance <-> EtherCAT Master EJxxxx/Beckhoff EJ7xxx/A_0008(EJ7342-0000-0020)
//     PlcTask Inputs/GVL_iXlinker.EtherCAT_Master_EJxxxx.Beckhoff_EJ7xxx.A_0008_EJ7342_0000_0020.ENC_Status_compact_Channel_1.Status/Latch_extern_valid <-> ENC Status compact Channel 1/Status/Latch extern valid
//     PlcTask Inputs/GVL_iXlinker.EtherCAT_Master_EJxxxx.Beckhoff_EJ7xxx.A_0008_EJ7342_0000_0020.ENC_Status_compact_Channel_2.Status/Latch_extern_valid <-> ENC Status compact Channel 2/Status/Latch extern valid
//     PlcTask Inputs/GVL_iXlinker.EtherCAT_Master_EJxxxx.Beckhoff_EJ7xxx.A_0008_EJ7342_0000_0020.ENC_Status_compact_Channel_1.Status/Set_counter_done <-> ENC Status compact Channel 1/Status/Set counter done
//     PlcTask Inputs/GVL_iXlinker.EtherCAT_Master_EJxxxx.Beckhoff_EJ7xxx.A_0008_EJ7342_0000_0020.ENC_Status_compact_Channel_2.Status/Set_counter_done <-> ENC Status compact Channel 2/Status/Set counter done
//     PlcTask Inputs/GVL_iXlinker.EtherCAT_Master_EJxxxx.Beckhoff_EJ7xxx.A_0008_EJ7342_0000_0020.ENC_Status_compact_Channel_1.Status/Counter_underflow <-> ENC Status compact Channel 1/Status/Counter underflow
//     PlcTask Inputs/GVL_iXlinker.EtherCAT_Master_EJxxxx.Beckhoff_EJ7xxx.A_0008_EJ7342_0000_0020.ENC_Status_compact_Channel_2.Status/Counter_underflow <-> ENC Status compact Channel 2/Status/Counter underflow
//     PlcTask Inputs/GVL_iXlinker.EtherCAT_Master_EJxxxx.Beckhoff_EJ7xxx.A_0008_EJ7342_0000_0020.ENC_Status_compact_Channel_1.Status/Counter_overflow <-> ENC Status compact Channel 1/Status/Counter overflow
//     PlcTask Inputs/GVL_iXlinker.EtherCAT_Master_EJxxxx.Beckhoff_EJ7xxx.A_0008_EJ7342_0000_0020.ENC_Status_compact_Channel_2.Status/Counter_overflow <-> ENC Status compact Channel 2/Status/Counter overflow
//     PlcTask Inputs/GVL_iXlinker.EtherCAT_Master_EJxxxx.Beckhoff_EJ7xxx.A_0008_EJ7342_0000_0020.ENC_Status_compact_Channel_1.Status/Extrapolation_stall <-> ENC Status compact Channel 1/Status/Extrapolation stall
//     PlcTask Inputs/GVL_iXlinker.EtherCAT_Master_EJxxxx.Beckhoff_EJ7xxx.A_0008_EJ7342_0000_0020.ENC_Status_compact_Channel_2.Status/Extrapolation_stall <-> ENC Status compact Channel 2/Status/Extrapolation stall
//     PlcTask Inputs/GVL_iXlinker.EtherCAT_Master_EJxxxx.Beckhoff_EJ7xxx.A_0008_EJ7342_0000_0020.ENC_Status_compact_Channel_1.Status/Status_of_input_A <-> ENC Status compact Channel 1/Status/Status of input A
//     PlcTask Inputs/GVL_iXlinker.EtherCAT_Master_EJxxxx.Beckhoff_EJ7xxx.A_0008_EJ7342_0000_0020.ENC_Status_compact_Channel_2.Status/Status_of_input_A <-> ENC Status compact Channel 2/Status/Status of input A
//     PlcTask Inputs/GVL_iXlinker.EtherCAT_Master_EJxxxx.Beckhoff_EJ7xxx.A_0008_EJ7342_0000_0020.ENC_Status_compact_Channel_1.Status/Status_of_input_B <-> ENC Status compact Channel 1/Status/Status of input B
//     PlcTask Inputs/GVL_iXlinker.EtherCAT_Master_EJxxxx.Beckhoff_EJ7xxx.A_0008_EJ7342_0000_0020.ENC_Status_compact_Channel_2.Status/Status_of_input_B <-> ENC Status compact Channel 2/Status/Status of input B
//     PlcTask Inputs/GVL_iXlinker.EtherCAT_Master_EJxxxx.Beckhoff_EJ7xxx.A_0008_EJ7342_0000_0020.ENC_Status_compact_Channel_1.Status/Status_of_extern_latch <-> ENC Status compact Channel 1/Status/Status of extern latch
//     PlcTask Inputs/GVL_iXlinker.EtherCAT_Master_EJxxxx.Beckhoff_EJ7xxx.A_0008_EJ7342_0000_0020.ENC_Status_compact_Channel_2.Status/Status_of_extern_latch <-> ENC Status compact Channel 2/Status/Status of extern latch
//     PlcTask Inputs/GVL_iXlinker.EtherCAT_Master_EJxxxx.Beckhoff_EJ7xxx.A_0008_EJ7342_0000_0020.ENC_Status_compact_Channel_1.Status/Sync_error <-> ENC Status compact Channel 1/Status/Sync error
//     PlcTask Inputs/GVL_iXlinker.EtherCAT_Master_EJxxxx.Beckhoff_EJ7xxx.A_0008_EJ7342_0000_0020.ENC_Status_compact_Channel_2.Status/Sync_error <-> ENC Status compact Channel 2/Status/Sync error
//     PlcTask Inputs/GVL_iXlinker.EtherCAT_Master_EJxxxx.Beckhoff_EJ7xxx.A_0008_EJ7342_0000_0020.ENC_Status_compact_Channel_1.Status/TxPDO_Toggle <-> ENC Status compact Channel 1/Status/TxPDO Toggle
//     PlcTask Inputs/GVL_iXlinker.EtherCAT_Master_EJxxxx.Beckhoff_EJ7xxx.A_0008_EJ7342_0000_0020.ENC_Status_compact_Channel_2.Status/TxPDO_Toggle <-> ENC Status compact Channel 2/Status/TxPDO Toggle
//     PlcTask Inputs/GVL_iXlinker.EtherCAT_Master_EJxxxx.Beckhoff_EJ7xxx.A_0008_EJ7342_0000_0020.ENC_Status_compact_Channel_1.Counter_value <-> ENC Status compact Channel 1/Counter value
//     PlcTask Inputs/GVL_iXlinker.EtherCAT_Master_EJxxxx.Beckhoff_EJ7xxx.A_0008_EJ7342_0000_0020.ENC_Status_compact_Channel_2.Counter_value <-> ENC Status compact Channel 2/Counter value
//     PlcTask Inputs/GVL_iXlinker.EtherCAT_Master_EJxxxx.Beckhoff_EJ7xxx.A_0008_EJ7342_0000_0020.ENC_Status_compact_Channel_1.Latch_value <-> ENC Status compact Channel 1/Latch value
//     PlcTask Inputs/GVL_iXlinker.EtherCAT_Master_EJxxxx.Beckhoff_EJ7xxx.A_0008_EJ7342_0000_0020.ENC_Status_compact_Channel_2.Latch_value <-> ENC Status compact Channel 2/Latch value
//     PlcTask Inputs/GVL_iXlinker.EtherCAT_Master_EJxxxx.Beckhoff_EJ7xxx.A_0008_EJ7342_0000_0020.DCM_Status_Channel_1.Status/Ready_to_enable <-> DCM Status Channel 1/Status/Ready to enable
//     PlcTask Inputs/GVL_iXlinker.EtherCAT_Master_EJxxxx.Beckhoff_EJ7xxx.A_0008_EJ7342_0000_0020.DCM_Status_Channel_2.Status/Ready_to_enable <-> DCM Status Channel 2/Status/Ready to enable
//     PlcTask Inputs/GVL_iXlinker.EtherCAT_Master_EJxxxx.Beckhoff_EJ7xxx.A_0008_EJ7342_0000_0020.DCM_Status_Channel_1.Status/Ready <-> DCM Status Channel 1/Status/Ready
//     PlcTask Inputs/GVL_iXlinker.EtherCAT_Master_EJxxxx.Beckhoff_EJ7xxx.A_0008_EJ7342_0000_0020.DCM_Status_Channel_2.Status/Ready <-> DCM Status Channel 2/Status/Ready
//     PlcTask Inputs/GVL_iXlinker.EtherCAT_Master_EJxxxx.Beckhoff_EJ7xxx.A_0008_EJ7342_0000_0020.DCM_Status_Channel_1.Status/Warning <-> DCM Status Channel 1/Status/Warning
//     PlcTask Inputs/GVL_iXlinker.EtherCAT_Master_EJxxxx.Beckhoff_EJ7xxx.A_0008_EJ7342_0000_0020.DCM_Status_Channel_2.Status/Warning <-> DCM Status Channel 2/Status/Warning
//     PlcTask Inputs/GVL_iXlinker.EtherCAT_Master_EJxxxx.Beckhoff_EJ7xxx.A_0008_EJ7342_0000_0020.DCM_Status_Channel_1.Status/Error <-> DCM Status Channel 1/Status/Error
//     PlcTask Inputs/GVL_iXlinker.EtherCAT_Master_EJxxxx.Beckhoff_EJ7xxx.A_0008_EJ7342_0000_0020.DCM_Status_Channel_2.Status/Error <-> DCM Status Channel 2/Status/Error
//     PlcTask Inputs/GVL_iXlinker.EtherCAT_Master_EJxxxx.Beckhoff_EJ7xxx.A_0008_EJ7342_0000_0020.DCM_Status_Channel_1.Status/Moving_positive <-> DCM Status Channel 1/Status/Moving positive
//     PlcTask Inputs/GVL_iXlinker.EtherCAT_Master_EJxxxx.Beckhoff_EJ7xxx.A_0008_EJ7342_0000_0020.DCM_Status_Channel_2.Status/Moving_positive <-> DCM Status Channel 2/Status/Moving positive
//     PlcTask Inputs/GVL_iXlinker.EtherCAT_Master_EJxxxx.Beckhoff_EJ7xxx.A_0008_EJ7342_0000_0020.DCM_Status_Channel_1.Status/Moving_negative <-> DCM Status Channel 1/Status/Moving negative
//     PlcTask Inputs/GVL_iXlinker.EtherCAT_Master_EJxxxx.Beckhoff_EJ7xxx.A_0008_EJ7342_0000_0020.DCM_Status_Channel_2.Status/Moving_negative <-> DCM Status Channel 2/Status/Moving negative
//     PlcTask Inputs/GVL_iXlinker.EtherCAT_Master_EJxxxx.Beckhoff_EJ7xxx.A_0008_EJ7342_0000_0020.DCM_Status_Channel_1.Status/Torque_reduced <-> DCM Status Channel 1/Status/Torque reduced
//     PlcTask Inputs/GVL_iXlinker.EtherCAT_Master_EJxxxx.Beckhoff_EJ7xxx.A_0008_EJ7342_0000_0020.DCM_Status_Channel_2.Status/Torque_reduced <-> DCM Status Channel 2/Status/Torque reduced
//     PlcTask Inputs/GVL_iXlinker.EtherCAT_Master_EJxxxx.Beckhoff_EJ7xxx.A_0008_EJ7342_0000_0020.DCM_Status_Channel_1.Status/Digital_input_1 <-> DCM Status Channel 1/Status/Digital input 1
//     PlcTask Inputs/GVL_iXlinker.EtherCAT_Master_EJxxxx.Beckhoff_EJ7xxx.A_0008_EJ7342_0000_0020.DCM_Status_Channel_1.Status/Digital_input_2 <-> DCM Status Channel 1/Status/Digital input 2
//     PlcTask Inputs/GVL_iXlinker.EtherCAT_Master_EJxxxx.Beckhoff_EJ7xxx.A_0008_EJ7342_0000_0020.DCM_Status_Channel_2.Status/Digital_input_1 <-> DCM Status Channel 2/Status/Digital input 1
//     PlcTask Inputs/GVL_iXlinker.EtherCAT_Master_EJxxxx.Beckhoff_EJ7xxx.A_0008_EJ7342_0000_0020.DCM_Status_Channel_2.Status/Digital_input_2 <-> DCM Status Channel 2/Status/Digital input 2
//     PlcTask Inputs/GVL_iXlinker.EtherCAT_Master_EJxxxx.Beckhoff_EJ7xxx.A_0008_EJ7342_0000_0020.DCM_Status_Channel_1.Status/Sync_error <-> DCM Status Channel 1/Status/Sync error
//     PlcTask Inputs/GVL_iXlinker.EtherCAT_Master_EJxxxx.Beckhoff_EJ7xxx.A_0008_EJ7342_0000_0020.DCM_Status_Channel_2.Status/Sync_error <-> DCM Status Channel 2/Status/Sync error
//     PlcTask Inputs/GVL_iXlinker.EtherCAT_Master_EJxxxx.Beckhoff_EJ7xxx.A_0008_EJ7342_0000_0020.DCM_Status_Channel_1.Status/TxPDO_Toggle <-> DCM Status Channel 1/Status/TxPDO Toggle
//     PlcTask Inputs/GVL_iXlinker.EtherCAT_Master_EJxxxx.Beckhoff_EJ7xxx.A_0008_EJ7342_0000_0020.DCM_Status_Channel_2.Status/TxPDO_Toggle <-> DCM Status Channel 2/Status/TxPDO Toggle
//     PlcTask Outputs/GVL_iXlinker.EtherCAT_Master_EJxxxx.Beckhoff_EJ7xxx.A_0008_EJ7342_0000_0020.ENC_Control_compact_Channel_1.Control/Enable_latch_extern_on_positive_edge <-> ENC Control compact Channel 1/Control/Enable latch extern on positive edge
//     PlcTask Outputs/GVL_iXlinker.EtherCAT_Master_EJxxxx.Beckhoff_EJ7xxx.A_0008_EJ7342_0000_0020.ENC_Control_compact_Channel_2.Control/Enable_latch_extern_on_positive_edge <-> ENC Control compact Channel 2/Control/Enable latch extern on positive edge
//     PlcTask Outputs/GVL_iXlinker.EtherCAT_Master_EJxxxx.Beckhoff_EJ7xxx.A_0008_EJ7342_0000_0020.ENC_Control_compact_Channel_1.Control/Set_counter <-> ENC Control compact Channel 1/Control/Set counter
//     PlcTask Outputs/GVL_iXlinker.EtherCAT_Master_EJxxxx.Beckhoff_EJ7xxx.A_0008_EJ7342_0000_0020.ENC_Control_compact_Channel_2.Control/Set_counter <-> ENC Control compact Channel 2/Control/Set counter
//     PlcTask Outputs/GVL_iXlinker.EtherCAT_Master_EJxxxx.Beckhoff_EJ7xxx.A_0008_EJ7342_0000_0020.ENC_Control_compact_Channel_1.Control/Enable_latch_extern_on_negative_edge <-> ENC Control compact Channel 1/Control/Enable latch extern on negative edge
//     PlcTask Outputs/GVL_iXlinker.EtherCAT_Master_EJxxxx.Beckhoff_EJ7xxx.A_0008_EJ7342_0000_0020.ENC_Control_compact_Channel_2.Control/Enable_latch_extern_on_negative_edge <-> ENC Control compact Channel 2/Control/Enable latch extern on negative edge
//     PlcTask Outputs/GVL_iXlinker.EtherCAT_Master_EJxxxx.Beckhoff_EJ7xxx.A_0008_EJ7342_0000_0020.ENC_Control_compact_Channel_1.Set_counter_value <-> ENC Control compact Channel 1/Set counter value
//     PlcTask Outputs/GVL_iXlinker.EtherCAT_Master_EJxxxx.Beckhoff_EJ7xxx.A_0008_EJ7342_0000_0020.ENC_Control_compact_Channel_2.Set_counter_value <-> ENC Control compact Channel 2/Set counter value
//     PlcTask Outputs/GVL_iXlinker.EtherCAT_Master_EJxxxx.Beckhoff_EJ7xxx.A_0008_EJ7342_0000_0020.DCM_Control_Channel_1.Control/Enable <-> DCM Control Channel 1/Control/Enable
//     PlcTask Outputs/GVL_iXlinker.EtherCAT_Master_EJxxxx.Beckhoff_EJ7xxx.A_0008_EJ7342_0000_0020.DCM_Control_Channel_2.Control/Enable <-> DCM Control Channel 2/Control/Enable
//     PlcTask Outputs/GVL_iXlinker.EtherCAT_Master_EJxxxx.Beckhoff_EJ7xxx.A_0008_EJ7342_0000_0020.DCM_Control_Channel_1.Control/Reset <-> DCM Control Channel 1/Control/Reset
//     PlcTask Outputs/GVL_iXlinker.EtherCAT_Master_EJxxxx.Beckhoff_EJ7xxx.A_0008_EJ7342_0000_0020.DCM_Control_Channel_2.Control/Reset <-> DCM Control Channel 2/Control/Reset
//     PlcTask Outputs/GVL_iXlinker.EtherCAT_Master_EJxxxx.Beckhoff_EJ7xxx.A_0008_EJ7342_0000_0020.DCM_Control_Channel_1.Control/Reduce_torque <-> DCM Control Channel 1/Control/Reduce torque
//     PlcTask Outputs/GVL_iXlinker.EtherCAT_Master_EJxxxx.Beckhoff_EJ7xxx.A_0008_EJ7342_0000_0020.DCM_Control_Channel_2.Control/Reduce_torque <-> DCM Control Channel 2/Control/Reduce torque
//     PlcTask Outputs/GVL_iXlinker.EtherCAT_Master_EJxxxx.Beckhoff_EJ7xxx.A_0008_EJ7342_0000_0020.DCM_Velocity_Channel_1.Velocity <-> DCM Velocity Channel 1/Velocity
//     PlcTask Outputs/GVL_iXlinker.EtherCAT_Master_EJxxxx.Beckhoff_EJ7xxx.A_0008_EJ7342_0000_0020.DCM_Velocity_Channel_2.Velocity <-> DCM Velocity Channel 2/Velocity
//     PlcTask Inputs/GVL_iXlinker.EtherCAT_Master_EJxxxx.Beckhoff_EJ7xxx.A_0008_EJ7342_0000_0020.WcState.WcState <-> WcState/WcState
//     PlcTask Inputs/GVL_iXlinker.EtherCAT_Master_EJxxxx.Beckhoff_EJ7xxx.A_0008_EJ7342_0000_0020.WcState.InputToggle <-> WcState/InputToggle
//     PlcTask Inputs/GVL_iXlinker.EtherCAT_Master_EJxxxx.Beckhoff_EJ7xxx.A_0008_EJ7342_0000_0020.InfoData.AdsAddr <-> InfoData/AdsAddr
//     PlcTask Inputs/GVL_iXlinker.EtherCAT_Master_EJxxxx.Beckhoff_EJ7xxx.A_0008_EJ7342_0000_0020.InfoData.Chn0 <-> InfoData/Chn0
//     PlcTask Inputs/GVL_iXlinker.EtherCAT_Master_EJxxxx.Beckhoff_EJ7xxx.A_0008_EJ7342_0000_0020.InfoData.Chn1 <-> InfoData/Chn1
//     PlcTask Inputs/GVL_iXlinker.EtherCAT_Master_EJxxxx.Beckhoff_EJ7xxx.A_0008_EJ7342_0000_0020.InfoData.Chn2 <-> InfoData/Chn2
//     PlcTask Inputs/GVL_iXlinker.EtherCAT_Master_EJxxxx.Beckhoff_EJ7xxx.A_0008_EJ7342_0000_0020.InfoData.Chn3 <-> InfoData/Chn3
//     PlcTask Inputs/GVL_iXlinker.EtherCAT_Master_EJxxxx.Beckhoff_EJ7xxx.A_0008_EJ7342_0000_0020.InfoData.State <-> InfoData/State
//   PLC/PLC Instance <-> EtherCAT Master EJxxxx/Beckhoff EJ7xxx/A_0009(EJ7211-0010-0026)
//     PlcTask Inputs/GVL_iXlinker.EtherCAT_Master_EJxxxx.Beckhoff_EJ7xxx.A_0009_EJ7211_0010_0026.FB_Position.Position <-> FB Position/Position
//     PlcTask Inputs/GVL_iXlinker.EtherCAT_Master_EJxxxx.Beckhoff_EJ7xxx.A_0009_EJ7211_0010_0026.DRV_Statusword.Statusword <-> DRV Statusword/Statusword
//     PlcTask Outputs/GVL_iXlinker.EtherCAT_Master_EJxxxx.Beckhoff_EJ7xxx.A_0009_EJ7211_0010_0026.DRV_Controlword.Controlword <-> DRV Controlword/Controlword
//     PlcTask Outputs/GVL_iXlinker.EtherCAT_Master_EJxxxx.Beckhoff_EJ7xxx.A_0009_EJ7211_0010_0026.DRV_Target_velocity.Target_velocity <-> DRV Target velocity/Target velocity
//     PlcTask Inputs/GVL_iXlinker.EtherCAT_Master_EJxxxx.Beckhoff_EJ7xxx.A_0009_EJ7211_0010_0026.WcState.WcState <-> WcState/WcState
//     PlcTask Inputs/GVL_iXlinker.EtherCAT_Master_EJxxxx.Beckhoff_EJ7xxx.A_0009_EJ7211_0010_0026.WcState.InputToggle <-> WcState/InputToggle
//     PlcTask Inputs/GVL_iXlinker.EtherCAT_Master_EJxxxx.Beckhoff_EJ7xxx.A_0009_EJ7211_0010_0026.InfoData.AdsAddr <-> InfoData/AdsAddr
//     PlcTask Inputs/GVL_iXlinker.EtherCAT_Master_EJxxxx.Beckhoff_EJ7xxx.A_0009_EJ7211_0010_0026.InfoData.DcOutputShift <-> InfoData/DcOutputShift
//     PlcTask Inputs/GVL_iXlinker.EtherCAT_Master_EJxxxx.Beckhoff_EJ7xxx.A_0009_EJ7211_0010_0026.InfoData.DcInputShift <-> InfoData/DcInputShift
//     PlcTask Inputs/GVL_iXlinker.EtherCAT_Master_EJxxxx.Beckhoff_EJ7xxx.A_0009_EJ7211_0010_0026.InfoData.Chn0 <-> InfoData/Chn0
//     PlcTask Inputs/GVL_iXlinker.EtherCAT_Master_EJxxxx.Beckhoff_EJ7xxx.A_0009_EJ7211_0010_0026.InfoData.State <-> InfoData/State
//   PLC/PLC Instance <-> EtherCAT Master EJxxxx/Beckhoff EJ7xxx/A_0010(EJ7211-0010-0027)
//     PlcTask Inputs/GVL_iXlinker.EtherCAT_Master_EJxxxx.Beckhoff_EJ7xxx.A_0010_EJ7211_0010_0027.FB_Position.Position <-> FB Position/Position
//     PlcTask Inputs/GVL_iXlinker.EtherCAT_Master_EJxxxx.Beckhoff_EJ7xxx.A_0010_EJ7211_0010_0027.DRV_Statusword.Statusword <-> DRV Statusword/Statusword
//     PlcTask Outputs/GVL_iXlinker.EtherCAT_Master_EJxxxx.Beckhoff_EJ7xxx.A_0010_EJ7211_0010_0027.DRV_Controlword.Controlword <-> DRV Controlword/Controlword
//     PlcTask Outputs/GVL_iXlinker.EtherCAT_Master_EJxxxx.Beckhoff_EJ7xxx.A_0010_EJ7211_0010_0027.DRV_Target_velocity.Target_velocity <-> DRV Target velocity/Target velocity
//     PlcTask Inputs/GVL_iXlinker.EtherCAT_Master_EJxxxx.Beckhoff_EJ7xxx.A_0010_EJ7211_0010_0027.WcState.WcState <-> WcState/WcState
//     PlcTask Inputs/GVL_iXlinker.EtherCAT_Master_EJxxxx.Beckhoff_EJ7xxx.A_0010_EJ7211_0010_0027.WcState.InputToggle <-> WcState/InputToggle
//     PlcTask Inputs/GVL_iXlinker.EtherCAT_Master_EJxxxx.Beckhoff_EJ7xxx.A_0010_EJ7211_0010_0027.InfoData.AdsAddr <-> InfoData/AdsAddr
//     PlcTask Inputs/GVL_iXlinker.EtherCAT_Master_EJxxxx.Beckhoff_EJ7xxx.A_0010_EJ7211_0010_0027.InfoData.DcOutputShift <-> InfoData/DcOutputShift
//     PlcTask Inputs/GVL_iXlinker.EtherCAT_Master_EJxxxx.Beckhoff_EJ7xxx.A_0010_EJ7211_0010_0027.InfoData.DcInputShift <-> InfoData/DcInputShift
//     PlcTask Inputs/GVL_iXlinker.EtherCAT_Master_EJxxxx.Beckhoff_EJ7xxx.A_0010_EJ7211_0010_0027.InfoData.Chn0 <-> InfoData/Chn0
//     PlcTask Inputs/GVL_iXlinker.EtherCAT_Master_EJxxxx.Beckhoff_EJ7xxx.A_0010_EJ7211_0010_0027.InfoData.State <-> InfoData/State
//   PLC/PLC Instance <-> EtherCAT Master EJxxxx/Beckhoff EJ7xxx/A_0011(EJ7211-0010-0028)
//     PlcTask Inputs/GVL_iXlinker.EtherCAT_Master_EJxxxx.Beckhoff_EJ7xxx.A_0011_EJ7211_0010_0028.FB_Position.Position <-> FB Position/Position
//     PlcTask Inputs/GVL_iXlinker.EtherCAT_Master_EJxxxx.Beckhoff_EJ7xxx.A_0011_EJ7211_0010_0028.DRV_Statusword.Statusword <-> DRV Statusword/Statusword
//     PlcTask Outputs/GVL_iXlinker.EtherCAT_Master_EJxxxx.Beckhoff_EJ7xxx.A_0011_EJ7211_0010_0028.DRV_Controlword.Controlword <-> DRV Controlword/Controlword
//     PlcTask Outputs/GVL_iXlinker.EtherCAT_Master_EJxxxx.Beckhoff_EJ7xxx.A_0011_EJ7211_0010_0028.DRV_Target_velocity.Target_velocity <-> DRV Target velocity/Target velocity
//     PlcTask Inputs/GVL_iXlinker.EtherCAT_Master_EJxxxx.Beckhoff_EJ7xxx.A_0011_EJ7211_0010_0028.WcState.WcState <-> WcState/WcState
//     PlcTask Inputs/GVL_iXlinker.EtherCAT_Master_EJxxxx.Beckhoff_EJ7xxx.A_0011_EJ7211_0010_0028.WcState.InputToggle <-> WcState/InputToggle
//     PlcTask Inputs/GVL_iXlinker.EtherCAT_Master_EJxxxx.Beckhoff_EJ7xxx.A_0011_EJ7211_0010_0028.InfoData.AdsAddr <-> InfoData/AdsAddr
//     PlcTask Inputs/GVL_iXlinker.EtherCAT_Master_EJxxxx.Beckhoff_EJ7xxx.A_0011_EJ7211_0010_0028.InfoData.DcOutputShift <-> InfoData/DcOutputShift
//     PlcTask Inputs/GVL_iXlinker.EtherCAT_Master_EJxxxx.Beckhoff_EJ7xxx.A_0011_EJ7211_0010_0028.InfoData.DcInputShift <-> InfoData/DcInputShift
//     PlcTask Inputs/GVL_iXlinker.EtherCAT_Master_EJxxxx.Beckhoff_EJ7xxx.A_0011_EJ7211_0010_0028.InfoData.Chn0 <-> InfoData/Chn0
//     PlcTask Inputs/GVL_iXlinker.EtherCAT_Master_EJxxxx.Beckhoff_EJ7xxx.A_0011_EJ7211_0010_0028.InfoData.State <-> InfoData/State
//   PLC/PLC Instance <-> EtherCAT Master EJxxxx/Beckhoff EJ7xxx/A_0012(EJ7211-0010-0029)
//     PlcTask Inputs/GVL_iXlinker.EtherCAT_Master_EJxxxx.Beckhoff_EJ7xxx.A_0012_EJ7211_0010_0029.FB_Position.Position <-> FB Position/Position
//     PlcTask Inputs/GVL_iXlinker.EtherCAT_Master_EJxxxx.Beckhoff_EJ7xxx.A_0012_EJ7211_0010_0029.DRV_Statusword.Statusword <-> DRV Statusword/Statusword
//     PlcTask Outputs/GVL_iXlinker.EtherCAT_Master_EJxxxx.Beckhoff_EJ7xxx.A_0012_EJ7211_0010_0029.DRV_Controlword.Controlword <-> DRV Controlword/Controlword
//     PlcTask Outputs/GVL_iXlinker.EtherCAT_Master_EJxxxx.Beckhoff_EJ7xxx.A_0012_EJ7211_0010_0029.DRV_Target_velocity.Target_velocity <-> DRV Target velocity/Target velocity
//     PlcTask Inputs/GVL_iXlinker.EtherCAT_Master_EJxxxx.Beckhoff_EJ7xxx.A_0012_EJ7211_0010_0029.WcState.WcState <-> WcState/WcState
//     PlcTask Inputs/GVL_iXlinker.EtherCAT_Master_EJxxxx.Beckhoff_EJ7xxx.A_0012_EJ7211_0010_0029.WcState.InputToggle <-> WcState/InputToggle
//     PlcTask Inputs/GVL_iXlinker.EtherCAT_Master_EJxxxx.Beckhoff_EJ7xxx.A_0012_EJ7211_0010_0029.InfoData.AdsAddr <-> InfoData/AdsAddr
//     PlcTask Inputs/GVL_iXlinker.EtherCAT_Master_EJxxxx.Beckhoff_EJ7xxx.A_0012_EJ7211_0010_0029.InfoData.DcOutputShift <-> InfoData/DcOutputShift
//     PlcTask Inputs/GVL_iXlinker.EtherCAT_Master_EJxxxx.Beckhoff_EJ7xxx.A_0012_EJ7211_0010_0029.InfoData.DcInputShift <-> InfoData/DcInputShift
//     PlcTask Inputs/GVL_iXlinker.EtherCAT_Master_EJxxxx.Beckhoff_EJ7xxx.A_0012_EJ7211_0010_0029.InfoData.Chn0 <-> InfoData/Chn0
//     PlcTask Inputs/GVL_iXlinker.EtherCAT_Master_EJxxxx.Beckhoff_EJ7xxx.A_0012_EJ7211_0010_0029.InfoData.State <-> InfoData/State
//   PLC/PLC Instance <-> EtherCAT Master EJxxxx/Beckhoff EJ7xxx/A_0013(EJ7211-0010-0030)
//     PlcTask Inputs/GVL_iXlinker.EtherCAT_Master_EJxxxx.Beckhoff_EJ7xxx.A_0013_EJ7211_0010_0030.FB_Position.Position <-> FB Position/Position
//     PlcTask Inputs/GVL_iXlinker.EtherCAT_Master_EJxxxx.Beckhoff_EJ7xxx.A_0013_EJ7211_0010_0030.DRV_Statusword.Statusword <-> DRV Statusword/Statusword
//     PlcTask Outputs/GVL_iXlinker.EtherCAT_Master_EJxxxx.Beckhoff_EJ7xxx.A_0013_EJ7211_0010_0030.DRV_Controlword.Controlword <-> DRV Controlword/Controlword
//     PlcTask Outputs/GVL_iXlinker.EtherCAT_Master_EJxxxx.Beckhoff_EJ7xxx.A_0013_EJ7211_0010_0030.DRV_Target_velocity.Target_velocity <-> DRV Target velocity/Target velocity
//     PlcTask Inputs/GVL_iXlinker.EtherCAT_Master_EJxxxx.Beckhoff_EJ7xxx.A_0013_EJ7211_0010_0030.WcState.WcState <-> WcState/WcState
//     PlcTask Inputs/GVL_iXlinker.EtherCAT_Master_EJxxxx.Beckhoff_EJ7xxx.A_0013_EJ7211_0010_0030.WcState.InputToggle <-> WcState/InputToggle
//     PlcTask Inputs/GVL_iXlinker.EtherCAT_Master_EJxxxx.Beckhoff_EJ7xxx.A_0013_EJ7211_0010_0030.InfoData.AdsAddr <-> InfoData/AdsAddr
//     PlcTask Inputs/GVL_iXlinker.EtherCAT_Master_EJxxxx.Beckhoff_EJ7xxx.A_0013_EJ7211_0010_0030.InfoData.DcOutputShift <-> InfoData/DcOutputShift
//     PlcTask Inputs/GVL_iXlinker.EtherCAT_Master_EJxxxx.Beckhoff_EJ7xxx.A_0013_EJ7211_0010_0030.InfoData.DcInputShift <-> InfoData/DcInputShift
//     PlcTask Inputs/GVL_iXlinker.EtherCAT_Master_EJxxxx.Beckhoff_EJ7xxx.A_0013_EJ7211_0010_0030.InfoData.Chn0 <-> InfoData/Chn0
//     PlcTask Inputs/GVL_iXlinker.EtherCAT_Master_EJxxxx.Beckhoff_EJ7xxx.A_0013_EJ7211_0010_0030.InfoData.Chn1 <-> InfoData/Chn1
//     PlcTask Inputs/GVL_iXlinker.EtherCAT_Master_EJxxxx.Beckhoff_EJ7xxx.A_0013_EJ7211_0010_0030.InfoData.State <-> InfoData/State
//   PLC/PLC Instance <-> EtherCAT Master EJxxxx/Beckhoff EJ7xxx/A_0014(EJ7211-0010-0031)
//     PlcTask Inputs/GVL_iXlinker.EtherCAT_Master_EJxxxx.Beckhoff_EJ7xxx.A_0014_EJ7211_0010_0031.FB_Position.Position <-> FB Position/Position
//     PlcTask Inputs/GVL_iXlinker.EtherCAT_Master_EJxxxx.Beckhoff_EJ7xxx.A_0014_EJ7211_0010_0031.DRV_Statusword.Statusword <-> DRV Statusword/Statusword
//     PlcTask Outputs/GVL_iXlinker.EtherCAT_Master_EJxxxx.Beckhoff_EJ7xxx.A_0014_EJ7211_0010_0031.DRV_Controlword.Controlword <-> DRV Controlword/Controlword
//     PlcTask Outputs/GVL_iXlinker.EtherCAT_Master_EJxxxx.Beckhoff_EJ7xxx.A_0014_EJ7211_0010_0031.DRV_Target_velocity.Target_velocity <-> DRV Target velocity/Target velocity
//     PlcTask Inputs/GVL_iXlinker.EtherCAT_Master_EJxxxx.Beckhoff_EJ7xxx.A_0014_EJ7211_0010_0031.WcState.WcState <-> WcState/WcState
//     PlcTask Inputs/GVL_iXlinker.EtherCAT_Master_EJxxxx.Beckhoff_EJ7xxx.A_0014_EJ7211_0010_0031.WcState.InputToggle <-> WcState/InputToggle
//     PlcTask Inputs/GVL_iXlinker.EtherCAT_Master_EJxxxx.Beckhoff_EJ7xxx.A_0014_EJ7211_0010_0031.InfoData.AdsAddr <-> InfoData/AdsAddr
//     PlcTask Inputs/GVL_iXlinker.EtherCAT_Master_EJxxxx.Beckhoff_EJ7xxx.A_0014_EJ7211_0010_0031.InfoData.DcOutputShift <-> InfoData/DcOutputShift
//     PlcTask Inputs/GVL_iXlinker.EtherCAT_Master_EJxxxx.Beckhoff_EJ7xxx.A_0014_EJ7211_0010_0031.InfoData.DcInputShift <-> InfoData/DcInputShift
//     PlcTask Inputs/GVL_iXlinker.EtherCAT_Master_EJxxxx.Beckhoff_EJ7xxx.A_0014_EJ7211_0010_0031.InfoData.Chn0 <-> InfoData/Chn0
//     PlcTask Inputs/GVL_iXlinker.EtherCAT_Master_EJxxxx.Beckhoff_EJ7xxx.A_0014_EJ7211_0010_0031.InfoData.Chn1 <-> InfoData/Chn1
//     PlcTask Inputs/GVL_iXlinker.EtherCAT_Master_EJxxxx.Beckhoff_EJ7xxx.A_0014_EJ7211_0010_0031.InfoData.State <-> InfoData/State
//   PLC/PLC Instance <-> EtherCAT Master EJxxxx/Beckhoff EJ7xxx/A_0015(EJ7211-0010-0032)
//     PlcTask Inputs/GVL_iXlinker.EtherCAT_Master_EJxxxx.Beckhoff_EJ7xxx.A_0015_EJ7211_0010_0032.FB_Position.Position <-> FB Position/Position
//     PlcTask Inputs/GVL_iXlinker.EtherCAT_Master_EJxxxx.Beckhoff_EJ7xxx.A_0015_EJ7211_0010_0032.DRV_Statusword.Statusword <-> DRV Statusword/Statusword
//     PlcTask Outputs/GVL_iXlinker.EtherCAT_Master_EJxxxx.Beckhoff_EJ7xxx.A_0015_EJ7211_0010_0032.DRV_Controlword.Controlword <-> DRV Controlword/Controlword
//     PlcTask Outputs/GVL_iXlinker.EtherCAT_Master_EJxxxx.Beckhoff_EJ7xxx.A_0015_EJ7211_0010_0032.DRV_Target_velocity.Target_velocity <-> DRV Target velocity/Target velocity
//     PlcTask Inputs/GVL_iXlinker.EtherCAT_Master_EJxxxx.Beckhoff_EJ7xxx.A_0015_EJ7211_0010_0032.WcState.WcState <-> WcState/WcState
//     PlcTask Inputs/GVL_iXlinker.EtherCAT_Master_EJxxxx.Beckhoff_EJ7xxx.A_0015_EJ7211_0010_0032.WcState.InputToggle <-> WcState/InputToggle
//     PlcTask Inputs/GVL_iXlinker.EtherCAT_Master_EJxxxx.Beckhoff_EJ7xxx.A_0015_EJ7211_0010_0032.InfoData.AdsAddr <-> InfoData/AdsAddr
//     PlcTask Inputs/GVL_iXlinker.EtherCAT_Master_EJxxxx.Beckhoff_EJ7xxx.A_0015_EJ7211_0010_0032.InfoData.DcOutputShift <-> InfoData/DcOutputShift
//     PlcTask Inputs/GVL_iXlinker.EtherCAT_Master_EJxxxx.Beckhoff_EJ7xxx.A_0015_EJ7211_0010_0032.InfoData.DcInputShift <-> InfoData/DcInputShift
//     PlcTask Inputs/GVL_iXlinker.EtherCAT_Master_EJxxxx.Beckhoff_EJ7xxx.A_0015_EJ7211_0010_0032.InfoData.Chn0 <-> InfoData/Chn0
//     PlcTask Inputs/GVL_iXlinker.EtherCAT_Master_EJxxxx.Beckhoff_EJ7xxx.A_0015_EJ7211_0010_0032.InfoData.Chn1 <-> InfoData/Chn1
//     PlcTask Inputs/GVL_iXlinker.EtherCAT_Master_EJxxxx.Beckhoff_EJ7xxx.A_0015_EJ7211_0010_0032.InfoData.State <-> InfoData/State
//   PLC/PLC Instance <-> EtherCAT Master EJxxxx/Beckhoff EJ7xxx/A_0016(EJ7211-0011-0026)
//     PlcTask Inputs/GVL_iXlinker.EtherCAT_Master_EJxxxx.Beckhoff_EJ7xxx.A_0016_EJ7211_0011_0026.DS402_Statusword.Statusword <-> DS402 Statusword/Statusword
//     PlcTask Inputs/GVL_iXlinker.EtherCAT_Master_EJxxxx.Beckhoff_EJ7xxx.A_0016_EJ7211_0011_0026.DS402_Position_actual_value.Position_actual_value <-> DS402 Position actual value/Position actual value
//     PlcTask Outputs/GVL_iXlinker.EtherCAT_Master_EJxxxx.Beckhoff_EJ7xxx.A_0016_EJ7211_0011_0026.DS402_Controlword.Controlword <-> DS402 Controlword/Controlword
//     PlcTask Outputs/GVL_iXlinker.EtherCAT_Master_EJxxxx.Beckhoff_EJ7xxx.A_0016_EJ7211_0011_0026.DS402_Target_velocity.Target_velocity <-> DS402 Target velocity/Target velocity
//     PlcTask Inputs/GVL_iXlinker.EtherCAT_Master_EJxxxx.Beckhoff_EJ7xxx.A_0016_EJ7211_0011_0026.WcState.WcState <-> WcState/WcState
//     PlcTask Inputs/GVL_iXlinker.EtherCAT_Master_EJxxxx.Beckhoff_EJ7xxx.A_0016_EJ7211_0011_0026.WcState.InputToggle <-> WcState/InputToggle
//     PlcTask Inputs/GVL_iXlinker.EtherCAT_Master_EJxxxx.Beckhoff_EJ7xxx.A_0016_EJ7211_0011_0026.InfoData.AdsAddr <-> InfoData/AdsAddr
//     PlcTask Inputs/GVL_iXlinker.EtherCAT_Master_EJxxxx.Beckhoff_EJ7xxx.A_0016_EJ7211_0011_0026.InfoData.DcOutputShift <-> InfoData/DcOutputShift
//     PlcTask Inputs/GVL_iXlinker.EtherCAT_Master_EJxxxx.Beckhoff_EJ7xxx.A_0016_EJ7211_0011_0026.InfoData.DcInputShift <-> InfoData/DcInputShift
//     PlcTask Inputs/GVL_iXlinker.EtherCAT_Master_EJxxxx.Beckhoff_EJ7xxx.A_0016_EJ7211_0011_0026.InfoData.Chn0 <-> InfoData/Chn0
//     PlcTask Inputs/GVL_iXlinker.EtherCAT_Master_EJxxxx.Beckhoff_EJ7xxx.A_0016_EJ7211_0011_0026.InfoData.State <-> InfoData/State
//   PLC/PLC Instance <-> EtherCAT Master EJxxxx/Beckhoff EJ7xxx/A_0017(EJ7211-0011-0027)
//     PlcTask Inputs/GVL_iXlinker.EtherCAT_Master_EJxxxx.Beckhoff_EJ7xxx.A_0017_EJ7211_0011_0027.DS402_Statusword.Statusword <-> DS402 Statusword/Statusword
//     PlcTask Inputs/GVL_iXlinker.EtherCAT_Master_EJxxxx.Beckhoff_EJ7xxx.A_0017_EJ7211_0011_0027.DS402_Position_actual_value.Position_actual_value <-> DS402 Position actual value/Position actual value
//     PlcTask Outputs/GVL_iXlinker.EtherCAT_Master_EJxxxx.Beckhoff_EJ7xxx.A_0017_EJ7211_0011_0027.DS402_Controlword.Controlword <-> DS402 Controlword/Controlword
//     PlcTask Outputs/GVL_iXlinker.EtherCAT_Master_EJxxxx.Beckhoff_EJ7xxx.A_0017_EJ7211_0011_0027.DS402_Target_velocity.Target_velocity <-> DS402 Target velocity/Target velocity
//     PlcTask Inputs/GVL_iXlinker.EtherCAT_Master_EJxxxx.Beckhoff_EJ7xxx.A_0017_EJ7211_0011_0027.WcState.WcState <-> WcState/WcState
//     PlcTask Inputs/GVL_iXlinker.EtherCAT_Master_EJxxxx.Beckhoff_EJ7xxx.A_0017_EJ7211_0011_0027.WcState.InputToggle <-> WcState/InputToggle
//     PlcTask Inputs/GVL_iXlinker.EtherCAT_Master_EJxxxx.Beckhoff_EJ7xxx.A_0017_EJ7211_0011_0027.InfoData.AdsAddr <-> InfoData/AdsAddr
//     PlcTask Inputs/GVL_iXlinker.EtherCAT_Master_EJxxxx.Beckhoff_EJ7xxx.A_0017_EJ7211_0011_0027.InfoData.DcOutputShift <-> InfoData/DcOutputShift
//     PlcTask Inputs/GVL_iXlinker.EtherCAT_Master_EJxxxx.Beckhoff_EJ7xxx.A_0017_EJ7211_0011_0027.InfoData.DcInputShift <-> InfoData/DcInputShift
//     PlcTask Inputs/GVL_iXlinker.EtherCAT_Master_EJxxxx.Beckhoff_EJ7xxx.A_0017_EJ7211_0011_0027.InfoData.Chn0 <-> InfoData/Chn0
//     PlcTask Inputs/GVL_iXlinker.EtherCAT_Master_EJxxxx.Beckhoff_EJ7xxx.A_0017_EJ7211_0011_0027.InfoData.State <-> InfoData/State
//   PLC/PLC Instance <-> EtherCAT Master EJxxxx/Beckhoff EJ7xxx/A_0018(EJ7211-0011-0028)
//     PlcTask Inputs/GVL_iXlinker.EtherCAT_Master_EJxxxx.Beckhoff_EJ7xxx.A_0018_EJ7211_0011_0028.DS402_Statusword.Statusword <-> DS402 Statusword/Statusword
//     PlcTask Inputs/GVL_iXlinker.EtherCAT_Master_EJxxxx.Beckhoff_EJ7xxx.A_0018_EJ7211_0011_0028.DS402_Position_actual_value.Position_actual_value <-> DS402 Position actual value/Position actual value
//     PlcTask Outputs/GVL_iXlinker.EtherCAT_Master_EJxxxx.Beckhoff_EJ7xxx.A_0018_EJ7211_0011_0028.DS402_Controlword.Controlword <-> DS402 Controlword/Controlword
//     PlcTask Outputs/GVL_iXlinker.EtherCAT_Master_EJxxxx.Beckhoff_EJ7xxx.A_0018_EJ7211_0011_0028.DS402_Target_velocity.Target_velocity <-> DS402 Target velocity/Target velocity
//     PlcTask Inputs/GVL_iXlinker.EtherCAT_Master_EJxxxx.Beckhoff_EJ7xxx.A_0018_EJ7211_0011_0028.WcState.WcState <-> WcState/WcState
//     PlcTask Inputs/GVL_iXlinker.EtherCAT_Master_EJxxxx.Beckhoff_EJ7xxx.A_0018_EJ7211_0011_0028.WcState.InputToggle <-> WcState/InputToggle
//     PlcTask Inputs/GVL_iXlinker.EtherCAT_Master_EJxxxx.Beckhoff_EJ7xxx.A_0018_EJ7211_0011_0028.InfoData.AdsAddr <-> InfoData/AdsAddr
//     PlcTask Inputs/GVL_iXlinker.EtherCAT_Master_EJxxxx.Beckhoff_EJ7xxx.A_0018_EJ7211_0011_0028.InfoData.DcOutputShift <-> InfoData/DcOutputShift
//     PlcTask Inputs/GVL_iXlinker.EtherCAT_Master_EJxxxx.Beckhoff_EJ7xxx.A_0018_EJ7211_0011_0028.InfoData.DcInputShift <-> InfoData/DcInputShift
//     PlcTask Inputs/GVL_iXlinker.EtherCAT_Master_EJxxxx.Beckhoff_EJ7xxx.A_0018_EJ7211_0011_0028.InfoData.Chn0 <-> InfoData/Chn0
//     PlcTask Inputs/GVL_iXlinker.EtherCAT_Master_EJxxxx.Beckhoff_EJ7xxx.A_0018_EJ7211_0011_0028.InfoData.State <-> InfoData/State
//   PLC/PLC Instance <-> EtherCAT Master EJxxxx/Beckhoff EJ7xxx/A_0019(EJ7211-0011-0029)
//     PlcTask Inputs/GVL_iXlinker.EtherCAT_Master_EJxxxx.Beckhoff_EJ7xxx.A_0019_EJ7211_0011_0029.DS402_Statusword.Statusword <-> DS402 Statusword/Statusword
//     PlcTask Inputs/GVL_iXlinker.EtherCAT_Master_EJxxxx.Beckhoff_EJ7xxx.A_0019_EJ7211_0011_0029.DS402_Position_actual_value.Position_actual_value <-> DS402 Position actual value/Position actual value
//     PlcTask Outputs/GVL_iXlinker.EtherCAT_Master_EJxxxx.Beckhoff_EJ7xxx.A_0019_EJ7211_0011_0029.DS402_Controlword.Controlword <-> DS402 Controlword/Controlword
//     PlcTask Outputs/GVL_iXlinker.EtherCAT_Master_EJxxxx.Beckhoff_EJ7xxx.A_0019_EJ7211_0011_0029.DS402_Target_velocity.Target_velocity <-> DS402 Target velocity/Target velocity
//     PlcTask Inputs/GVL_iXlinker.EtherCAT_Master_EJxxxx.Beckhoff_EJ7xxx.A_0019_EJ7211_0011_0029.WcState.WcState <-> WcState/WcState
//     PlcTask Inputs/GVL_iXlinker.EtherCAT_Master_EJxxxx.Beckhoff_EJ7xxx.A_0019_EJ7211_0011_0029.WcState.InputToggle <-> WcState/InputToggle
//     PlcTask Inputs/GVL_iXlinker.EtherCAT_Master_EJxxxx.Beckhoff_EJ7xxx.A_0019_EJ7211_0011_0029.InfoData.AdsAddr <-> InfoData/AdsAddr
//     PlcTask Inputs/GVL_iXlinker.EtherCAT_Master_EJxxxx.Beckhoff_EJ7xxx.A_0019_EJ7211_0011_0029.InfoData.DcOutputShift <-> InfoData/DcOutputShift
//     PlcTask Inputs/GVL_iXlinker.EtherCAT_Master_EJxxxx.Beckhoff_EJ7xxx.A_0019_EJ7211_0011_0029.InfoData.DcInputShift <-> InfoData/DcInputShift
//     PlcTask Inputs/GVL_iXlinker.EtherCAT_Master_EJxxxx.Beckhoff_EJ7xxx.A_0019_EJ7211_0011_0029.InfoData.Chn0 <-> InfoData/Chn0
//     PlcTask Inputs/GVL_iXlinker.EtherCAT_Master_EJxxxx.Beckhoff_EJ7xxx.A_0019_EJ7211_0011_0029.InfoData.State <-> InfoData/State
//   PLC/PLC Instance <-> EtherCAT Master EJxxxx/Beckhoff EJ7xxx/A_0020(EJ7211-0011-0030)
//     PlcTask Inputs/GVL_iXlinker.EtherCAT_Master_EJxxxx.Beckhoff_EJ7xxx.A_0020_EJ7211_0011_0030.DS402_Statusword.Statusword <-> DS402 Statusword/Statusword
//     PlcTask Inputs/GVL_iXlinker.EtherCAT_Master_EJxxxx.Beckhoff_EJ7xxx.A_0020_EJ7211_0011_0030.DS402_Position_actual_value.Position_actual_value <-> DS402 Position actual value/Position actual value
//     PlcTask Outputs/GVL_iXlinker.EtherCAT_Master_EJxxxx.Beckhoff_EJ7xxx.A_0020_EJ7211_0011_0030.DS402_Controlword.Controlword <-> DS402 Controlword/Controlword
//     PlcTask Outputs/GVL_iXlinker.EtherCAT_Master_EJxxxx.Beckhoff_EJ7xxx.A_0020_EJ7211_0011_0030.DS402_Target_velocity.Target_velocity <-> DS402 Target velocity/Target velocity
//     PlcTask Inputs/GVL_iXlinker.EtherCAT_Master_EJxxxx.Beckhoff_EJ7xxx.A_0020_EJ7211_0011_0030.WcState.WcState <-> WcState/WcState
//     PlcTask Inputs/GVL_iXlinker.EtherCAT_Master_EJxxxx.Beckhoff_EJ7xxx.A_0020_EJ7211_0011_0030.WcState.InputToggle <-> WcState/InputToggle
//     PlcTask Inputs/GVL_iXlinker.EtherCAT_Master_EJxxxx.Beckhoff_EJ7xxx.A_0020_EJ7211_0011_0030.InfoData.AdsAddr <-> InfoData/AdsAddr
//     PlcTask Inputs/GVL_iXlinker.EtherCAT_Master_EJxxxx.Beckhoff_EJ7xxx.A_0020_EJ7211_0011_0030.InfoData.DcOutputShift <-> InfoData/DcOutputShift
//     PlcTask Inputs/GVL_iXlinker.EtherCAT_Master_EJxxxx.Beckhoff_EJ7xxx.A_0020_EJ7211_0011_0030.InfoData.DcInputShift <-> InfoData/DcInputShift
//     PlcTask Inputs/GVL_iXlinker.EtherCAT_Master_EJxxxx.Beckhoff_EJ7xxx.A_0020_EJ7211_0011_0030.InfoData.Chn0 <-> InfoData/Chn0
//     PlcTask Inputs/GVL_iXlinker.EtherCAT_Master_EJxxxx.Beckhoff_EJ7xxx.A_0020_EJ7211_0011_0030.InfoData.State <-> InfoData/State
//   PLC/PLC Instance <-> EtherCAT Master EJxxxx/Beckhoff EJ7xxx/A_0021(EJ7211-0011-0031)
//     PlcTask Inputs/GVL_iXlinker.EtherCAT_Master_EJxxxx.Beckhoff_EJ7xxx.A_0021_EJ7211_0011_0031.DS402_Statusword.Statusword <-> DS402 Statusword/Statusword
//     PlcTask Inputs/GVL_iXlinker.EtherCAT_Master_EJxxxx.Beckhoff_EJ7xxx.A_0021_EJ7211_0011_0031.DS402_Position_actual_value.Position_actual_value <-> DS402 Position actual value/Position actual value
//     PlcTask Outputs/GVL_iXlinker.EtherCAT_Master_EJxxxx.Beckhoff_EJ7xxx.A_0021_EJ7211_0011_0031.DS402_Controlword.Controlword <-> DS402 Controlword/Controlword
//     PlcTask Outputs/GVL_iXlinker.EtherCAT_Master_EJxxxx.Beckhoff_EJ7xxx.A_0021_EJ7211_0011_0031.DS402_Target_velocity.Target_velocity <-> DS402 Target velocity/Target velocity
//     PlcTask Inputs/GVL_iXlinker.EtherCAT_Master_EJxxxx.Beckhoff_EJ7xxx.A_0021_EJ7211_0011_0031.WcState.WcState <-> WcState/WcState
//     PlcTask Inputs/GVL_iXlinker.EtherCAT_Master_EJxxxx.Beckhoff_EJ7xxx.A_0021_EJ7211_0011_0031.WcState.InputToggle <-> WcState/InputToggle
//     PlcTask Inputs/GVL_iXlinker.EtherCAT_Master_EJxxxx.Beckhoff_EJ7xxx.A_0021_EJ7211_0011_0031.InfoData.AdsAddr <-> InfoData/AdsAddr
//     PlcTask Inputs/GVL_iXlinker.EtherCAT_Master_EJxxxx.Beckhoff_EJ7xxx.A_0021_EJ7211_0011_0031.InfoData.DcOutputShift <-> InfoData/DcOutputShift
//     PlcTask Inputs/GVL_iXlinker.EtherCAT_Master_EJxxxx.Beckhoff_EJ7xxx.A_0021_EJ7211_0011_0031.InfoData.DcInputShift <-> InfoData/DcInputShift
//     PlcTask Inputs/GVL_iXlinker.EtherCAT_Master_EJxxxx.Beckhoff_EJ7xxx.A_0021_EJ7211_0011_0031.InfoData.Chn0 <-> InfoData/Chn0
//     PlcTask Inputs/GVL_iXlinker.EtherCAT_Master_EJxxxx.Beckhoff_EJ7xxx.A_0021_EJ7211_0011_0031.InfoData.State <-> InfoData/State
//   PLC/PLC Instance <-> EtherCAT Master EJxxxx/Beckhoff EJ7xxx/A_0022(EJ7211-0011-0032)
//     PlcTask Inputs/GVL_iXlinker.EtherCAT_Master_EJxxxx.Beckhoff_EJ7xxx.A_0022_EJ7211_0011_0032.DS402_Statusword.Statusword <-> DS402 Statusword/Statusword
//     PlcTask Inputs/GVL_iXlinker.EtherCAT_Master_EJxxxx.Beckhoff_EJ7xxx.A_0022_EJ7211_0011_0032.DS402_Position_actual_value.Position_actual_value <-> DS402 Position actual value/Position actual value
//     PlcTask Outputs/GVL_iXlinker.EtherCAT_Master_EJxxxx.Beckhoff_EJ7xxx.A_0022_EJ7211_0011_0032.DS402_Controlword.Controlword <-> DS402 Controlword/Controlword
//     PlcTask Outputs/GVL_iXlinker.EtherCAT_Master_EJxxxx.Beckhoff_EJ7xxx.A_0022_EJ7211_0011_0032.DS402_Target_velocity.Target_velocity <-> DS402 Target velocity/Target velocity
//     PlcTask Inputs/GVL_iXlinker.EtherCAT_Master_EJxxxx.Beckhoff_EJ7xxx.A_0022_EJ7211_0011_0032.WcState.WcState <-> WcState/WcState
//     PlcTask Inputs/GVL_iXlinker.EtherCAT_Master_EJxxxx.Beckhoff_EJ7xxx.A_0022_EJ7211_0011_0032.WcState.InputToggle <-> WcState/InputToggle
//     PlcTask Inputs/GVL_iXlinker.EtherCAT_Master_EJxxxx.Beckhoff_EJ7xxx.A_0022_EJ7211_0011_0032.InfoData.AdsAddr <-> InfoData/AdsAddr
//     PlcTask Inputs/GVL_iXlinker.EtherCAT_Master_EJxxxx.Beckhoff_EJ7xxx.A_0022_EJ7211_0011_0032.InfoData.DcOutputShift <-> InfoData/DcOutputShift
//     PlcTask Inputs/GVL_iXlinker.EtherCAT_Master_EJxxxx.Beckhoff_EJ7xxx.A_0022_EJ7211_0011_0032.InfoData.DcInputShift <-> InfoData/DcInputShift
//     PlcTask Inputs/GVL_iXlinker.EtherCAT_Master_EJxxxx.Beckhoff_EJ7xxx.A_0022_EJ7211_0011_0032.InfoData.Chn0 <-> InfoData/Chn0
//     PlcTask Inputs/GVL_iXlinker.EtherCAT_Master_EJxxxx.Beckhoff_EJ7xxx.A_0022_EJ7211_0011_0032.InfoData.State <-> InfoData/State
//   PLC/PLC Instance <-> EtherCAT Master EJxxxx/Beckhoff EJ7xxx/A_0023(EJ7211-9414-0029)
//     PlcTask Inputs/GVL_iXlinker.EtherCAT_Master_EJxxxx.Beckhoff_EJ7xxx.A_0023_EJ7211_9414_0029.FB_Position.Position <-> FB Position/Position
//     PlcTask Inputs/GVL_iXlinker.EtherCAT_Master_EJxxxx.Beckhoff_EJ7xxx.A_0023_EJ7211_9414_0029.DRV_Statusword.Statusword <-> DRV Statusword/Statusword
//     PlcTask Outputs/GVL_iXlinker.EtherCAT_Master_EJxxxx.Beckhoff_EJ7xxx.A_0023_EJ7211_9414_0029.DRV_Controlword.Controlword <-> DRV Controlword/Controlword
//     PlcTask Outputs/GVL_iXlinker.EtherCAT_Master_EJxxxx.Beckhoff_EJ7xxx.A_0023_EJ7211_9414_0029.DRV_Target_velocity.Target_velocity <-> DRV Target velocity/Target velocity
//     PlcTask Inputs/GVL_iXlinker.EtherCAT_Master_EJxxxx.Beckhoff_EJ7xxx.A_0023_EJ7211_9414_0029.WcState.WcState <-> WcState/WcState
//     PlcTask Inputs/GVL_iXlinker.EtherCAT_Master_EJxxxx.Beckhoff_EJ7xxx.A_0023_EJ7211_9414_0029.WcState.InputToggle <-> WcState/InputToggle
//     PlcTask Inputs/GVL_iXlinker.EtherCAT_Master_EJxxxx.Beckhoff_EJ7xxx.A_0023_EJ7211_9414_0029.InfoData.AdsAddr <-> InfoData/AdsAddr
//     PlcTask Inputs/GVL_iXlinker.EtherCAT_Master_EJxxxx.Beckhoff_EJ7xxx.A_0023_EJ7211_9414_0029.InfoData.DcOutputShift <-> InfoData/DcOutputShift
//     PlcTask Inputs/GVL_iXlinker.EtherCAT_Master_EJxxxx.Beckhoff_EJ7xxx.A_0023_EJ7211_9414_0029.InfoData.DcInputShift <-> InfoData/DcInputShift
//     PlcTask Inputs/GVL_iXlinker.EtherCAT_Master_EJxxxx.Beckhoff_EJ7xxx.A_0023_EJ7211_9414_0029.InfoData.Chn0 <-> InfoData/Chn0
//     PlcTask Inputs/GVL_iXlinker.EtherCAT_Master_EJxxxx.Beckhoff_EJ7xxx.A_0023_EJ7211_9414_0029.InfoData.State <-> InfoData/State
//   PLC/PLC Instance <-> EtherCAT Master EJxxxx/Beckhoff EJ7xxx/A_0024(EJ7211-9414-0030)
//     PlcTask Inputs/GVL_iXlinker.EtherCAT_Master_EJxxxx.Beckhoff_EJ7xxx.A_0024_EJ7211_9414_0030.FB_Position.Position <-> FB Position/Position
//     PlcTask Inputs/GVL_iXlinker.EtherCAT_Master_EJxxxx.Beckhoff_EJ7xxx.A_0024_EJ7211_9414_0030.DRV_Statusword.Statusword <-> DRV Statusword/Statusword
//     PlcTask Outputs/GVL_iXlinker.EtherCAT_Master_EJxxxx.Beckhoff_EJ7xxx.A_0024_EJ7211_9414_0030.DRV_Controlword.Controlword <-> DRV Controlword/Controlword
//     PlcTask Outputs/GVL_iXlinker.EtherCAT_Master_EJxxxx.Beckhoff_EJ7xxx.A_0024_EJ7211_9414_0030.DRV_Target_velocity.Target_velocity <-> DRV Target velocity/Target velocity
//     PlcTask Inputs/GVL_iXlinker.EtherCAT_Master_EJxxxx.Beckhoff_EJ7xxx.A_0024_EJ7211_9414_0030.WcState.WcState <-> WcState/WcState
//     PlcTask Inputs/GVL_iXlinker.EtherCAT_Master_EJxxxx.Beckhoff_EJ7xxx.A_0024_EJ7211_9414_0030.WcState.InputToggle <-> WcState/InputToggle
//     PlcTask Inputs/GVL_iXlinker.EtherCAT_Master_EJxxxx.Beckhoff_EJ7xxx.A_0024_EJ7211_9414_0030.InfoData.AdsAddr <-> InfoData/AdsAddr
//     PlcTask Inputs/GVL_iXlinker.EtherCAT_Master_EJxxxx.Beckhoff_EJ7xxx.A_0024_EJ7211_9414_0030.InfoData.DcOutputShift <-> InfoData/DcOutputShift
//     PlcTask Inputs/GVL_iXlinker.EtherCAT_Master_EJxxxx.Beckhoff_EJ7xxx.A_0024_EJ7211_9414_0030.InfoData.DcInputShift <-> InfoData/DcInputShift
//     PlcTask Inputs/GVL_iXlinker.EtherCAT_Master_EJxxxx.Beckhoff_EJ7xxx.A_0024_EJ7211_9414_0030.InfoData.Chn0 <-> InfoData/Chn0
//     PlcTask Inputs/GVL_iXlinker.EtherCAT_Master_EJxxxx.Beckhoff_EJ7xxx.A_0024_EJ7211_9414_0030.InfoData.Chn1 <-> InfoData/Chn1
//     PlcTask Inputs/GVL_iXlinker.EtherCAT_Master_EJxxxx.Beckhoff_EJ7xxx.A_0024_EJ7211_9414_0030.InfoData.Chn2 <-> InfoData/Chn2
//     PlcTask Inputs/GVL_iXlinker.EtherCAT_Master_EJxxxx.Beckhoff_EJ7xxx.A_0024_EJ7211_9414_0030.InfoData.State <-> InfoData/State
//   PLC/PLC Instance <-> EtherCAT Master EJxxxx/Beckhoff EJ7xxx/A_0025(EJ7211-9414-0031)
//     PlcTask Inputs/GVL_iXlinker.EtherCAT_Master_EJxxxx.Beckhoff_EJ7xxx.A_0025_EJ7211_9414_0031.FB_Position.Position <-> FB Position/Position
//     PlcTask Inputs/GVL_iXlinker.EtherCAT_Master_EJxxxx.Beckhoff_EJ7xxx.A_0025_EJ7211_9414_0031.DRV_Statusword.Statusword <-> DRV Statusword/Statusword
//     PlcTask Outputs/GVL_iXlinker.EtherCAT_Master_EJxxxx.Beckhoff_EJ7xxx.A_0025_EJ7211_9414_0031.DRV_Controlword.Controlword <-> DRV Controlword/Controlword
//     PlcTask Outputs/GVL_iXlinker.EtherCAT_Master_EJxxxx.Beckhoff_EJ7xxx.A_0025_EJ7211_9414_0031.DRV_Target_velocity.Target_velocity <-> DRV Target velocity/Target velocity
//     PlcTask Inputs/GVL_iXlinker.EtherCAT_Master_EJxxxx.Beckhoff_EJ7xxx.A_0025_EJ7211_9414_0031.WcState.WcState <-> WcState/WcState
//     PlcTask Inputs/GVL_iXlinker.EtherCAT_Master_EJxxxx.Beckhoff_EJ7xxx.A_0025_EJ7211_9414_0031.WcState.InputToggle <-> WcState/InputToggle
//     PlcTask Inputs/GVL_iXlinker.EtherCAT_Master_EJxxxx.Beckhoff_EJ7xxx.A_0025_EJ7211_9414_0031.InfoData.AdsAddr <-> InfoData/AdsAddr
//     PlcTask Inputs/GVL_iXlinker.EtherCAT_Master_EJxxxx.Beckhoff_EJ7xxx.A_0025_EJ7211_9414_0031.InfoData.DcOutputShift <-> InfoData/DcOutputShift
//     PlcTask Inputs/GVL_iXlinker.EtherCAT_Master_EJxxxx.Beckhoff_EJ7xxx.A_0025_EJ7211_9414_0031.InfoData.DcInputShift <-> InfoData/DcInputShift
//     PlcTask Inputs/GVL_iXlinker.EtherCAT_Master_EJxxxx.Beckhoff_EJ7xxx.A_0025_EJ7211_9414_0031.InfoData.Chn0 <-> InfoData/Chn0
//     PlcTask Inputs/GVL_iXlinker.EtherCAT_Master_EJxxxx.Beckhoff_EJ7xxx.A_0025_EJ7211_9414_0031.InfoData.Chn1 <-> InfoData/Chn1
//     PlcTask Inputs/GVL_iXlinker.EtherCAT_Master_EJxxxx.Beckhoff_EJ7xxx.A_0025_EJ7211_9414_0031.InfoData.Chn2 <-> InfoData/Chn2
//     PlcTask Inputs/GVL_iXlinker.EtherCAT_Master_EJxxxx.Beckhoff_EJ7xxx.A_0025_EJ7211_9414_0031.InfoData.State <-> InfoData/State
//   PLC/PLC Instance <-> EtherCAT Master EJxxxx/Beckhoff EJ7xxx/A_0026(EJ7211-9414-0032)
//     PlcTask Inputs/GVL_iXlinker.EtherCAT_Master_EJxxxx.Beckhoff_EJ7xxx.A_0026_EJ7211_9414_0032.FB_Position.Position <-> FB Position/Position
//     PlcTask Inputs/GVL_iXlinker.EtherCAT_Master_EJxxxx.Beckhoff_EJ7xxx.A_0026_EJ7211_9414_0032.DRV_Statusword.Statusword <-> DRV Statusword/Statusword
//     PlcTask Outputs/GVL_iXlinker.EtherCAT_Master_EJxxxx.Beckhoff_EJ7xxx.A_0026_EJ7211_9414_0032.DRV_Controlword.Controlword <-> DRV Controlword/Controlword
//     PlcTask Outputs/GVL_iXlinker.EtherCAT_Master_EJxxxx.Beckhoff_EJ7xxx.A_0026_EJ7211_9414_0032.DRV_Target_velocity.Target_velocity <-> DRV Target velocity/Target velocity
//     PlcTask Inputs/GVL_iXlinker.EtherCAT_Master_EJxxxx.Beckhoff_EJ7xxx.A_0026_EJ7211_9414_0032.WcState.WcState <-> WcState/WcState
//     PlcTask Inputs/GVL_iXlinker.EtherCAT_Master_EJxxxx.Beckhoff_EJ7xxx.A_0026_EJ7211_9414_0032.WcState.InputToggle <-> WcState/InputToggle
//     PlcTask Inputs/GVL_iXlinker.EtherCAT_Master_EJxxxx.Beckhoff_EJ7xxx.A_0026_EJ7211_9414_0032.InfoData.AdsAddr <-> InfoData/AdsAddr
//     PlcTask Inputs/GVL_iXlinker.EtherCAT_Master_EJxxxx.Beckhoff_EJ7xxx.A_0026_EJ7211_9414_0032.InfoData.DcOutputShift <-> InfoData/DcOutputShift
//     PlcTask Inputs/GVL_iXlinker.EtherCAT_Master_EJxxxx.Beckhoff_EJ7xxx.A_0026_EJ7211_9414_0032.InfoData.DcInputShift <-> InfoData/DcInputShift
//     PlcTask Inputs/GVL_iXlinker.EtherCAT_Master_EJxxxx.Beckhoff_EJ7xxx.A_0026_EJ7211_9414_0032.InfoData.Chn0 <-> InfoData/Chn0
//     PlcTask Inputs/GVL_iXlinker.EtherCAT_Master_EJxxxx.Beckhoff_EJ7xxx.A_0026_EJ7211_9414_0032.InfoData.Chn1 <-> InfoData/Chn1
//     PlcTask Inputs/GVL_iXlinker.EtherCAT_Master_EJxxxx.Beckhoff_EJ7xxx.A_0026_EJ7211_9414_0032.InfoData.Chn2 <-> InfoData/Chn2
//     PlcTask Inputs/GVL_iXlinker.EtherCAT_Master_EJxxxx.Beckhoff_EJ7xxx.A_0026_EJ7211_9414_0032.InfoData.State <-> InfoData/State
//   PLC/PLC Instance <-> EtherCAT Master EJxxxx/Beckhoff EJ7xxx/A_0027(EJ7211-9415-0029)
//     PlcTask Inputs/GVL_iXlinker.EtherCAT_Master_EJxxxx.Beckhoff_EJ7xxx.A_0027_EJ7211_9415_0029.DS402_Statusword.Statusword <-> DS402 Statusword/Statusword
//     PlcTask Inputs/GVL_iXlinker.EtherCAT_Master_EJxxxx.Beckhoff_EJ7xxx.A_0027_EJ7211_9415_0029.DS402_Position_actual_value.Position_actual_value <-> DS402 Position actual value/Position actual value
//     PlcTask Outputs/GVL_iXlinker.EtherCAT_Master_EJxxxx.Beckhoff_EJ7xxx.A_0027_EJ7211_9415_0029.DS402_Controlword.Controlword <-> DS402 Controlword/Controlword
//     PlcTask Outputs/GVL_iXlinker.EtherCAT_Master_EJxxxx.Beckhoff_EJ7xxx.A_0027_EJ7211_9415_0029.DS402_Target_velocity.Target_velocity <-> DS402 Target velocity/Target velocity
//     PlcTask Inputs/GVL_iXlinker.EtherCAT_Master_EJxxxx.Beckhoff_EJ7xxx.A_0027_EJ7211_9415_0029.WcState.WcState <-> WcState/WcState
//     PlcTask Inputs/GVL_iXlinker.EtherCAT_Master_EJxxxx.Beckhoff_EJ7xxx.A_0027_EJ7211_9415_0029.WcState.InputToggle <-> WcState/InputToggle
//     PlcTask Inputs/GVL_iXlinker.EtherCAT_Master_EJxxxx.Beckhoff_EJ7xxx.A_0027_EJ7211_9415_0029.InfoData.AdsAddr <-> InfoData/AdsAddr
//     PlcTask Inputs/GVL_iXlinker.EtherCAT_Master_EJxxxx.Beckhoff_EJ7xxx.A_0027_EJ7211_9415_0029.InfoData.DcOutputShift <-> InfoData/DcOutputShift
//     PlcTask Inputs/GVL_iXlinker.EtherCAT_Master_EJxxxx.Beckhoff_EJ7xxx.A_0027_EJ7211_9415_0029.InfoData.DcInputShift <-> InfoData/DcInputShift
//     PlcTask Inputs/GVL_iXlinker.EtherCAT_Master_EJxxxx.Beckhoff_EJ7xxx.A_0027_EJ7211_9415_0029.InfoData.Chn0 <-> InfoData/Chn0
//     PlcTask Inputs/GVL_iXlinker.EtherCAT_Master_EJxxxx.Beckhoff_EJ7xxx.A_0027_EJ7211_9415_0029.InfoData.State <-> InfoData/State
//   PLC/PLC Instance <-> EtherCAT Master EJxxxx/Beckhoff EJ7xxx/A_0028(EJ7211-9415-0030)
//     PlcTask Inputs/GVL_iXlinker.EtherCAT_Master_EJxxxx.Beckhoff_EJ7xxx.A_0028_EJ7211_9415_0030.DS402_Statusword.Statusword <-> DS402 Statusword/Statusword
//     PlcTask Inputs/GVL_iXlinker.EtherCAT_Master_EJxxxx.Beckhoff_EJ7xxx.A_0028_EJ7211_9415_0030.DS402_Position_actual_value.Position_actual_value <-> DS402 Position actual value/Position actual value
//     PlcTask Outputs/GVL_iXlinker.EtherCAT_Master_EJxxxx.Beckhoff_EJ7xxx.A_0028_EJ7211_9415_0030.DS402_Controlword.Controlword <-> DS402 Controlword/Controlword
//     PlcTask Outputs/GVL_iXlinker.EtherCAT_Master_EJxxxx.Beckhoff_EJ7xxx.A_0028_EJ7211_9415_0030.DS402_Target_velocity.Target_velocity <-> DS402 Target velocity/Target velocity
//     PlcTask Inputs/GVL_iXlinker.EtherCAT_Master_EJxxxx.Beckhoff_EJ7xxx.A_0028_EJ7211_9415_0030.WcState.WcState <-> WcState/WcState
//     PlcTask Inputs/GVL_iXlinker.EtherCAT_Master_EJxxxx.Beckhoff_EJ7xxx.A_0028_EJ7211_9415_0030.WcState.InputToggle <-> WcState/InputToggle
//     PlcTask Inputs/GVL_iXlinker.EtherCAT_Master_EJxxxx.Beckhoff_EJ7xxx.A_0028_EJ7211_9415_0030.InfoData.AdsAddr <-> InfoData/AdsAddr
//     PlcTask Inputs/GVL_iXlinker.EtherCAT_Master_EJxxxx.Beckhoff_EJ7xxx.A_0028_EJ7211_9415_0030.InfoData.DcOutputShift <-> InfoData/DcOutputShift
//     PlcTask Inputs/GVL_iXlinker.EtherCAT_Master_EJxxxx.Beckhoff_EJ7xxx.A_0028_EJ7211_9415_0030.InfoData.DcInputShift <-> InfoData/DcInputShift
//     PlcTask Inputs/GVL_iXlinker.EtherCAT_Master_EJxxxx.Beckhoff_EJ7xxx.A_0028_EJ7211_9415_0030.InfoData.Chn0 <-> InfoData/Chn0
//     PlcTask Inputs/GVL_iXlinker.EtherCAT_Master_EJxxxx.Beckhoff_EJ7xxx.A_0028_EJ7211_9415_0030.InfoData.State <-> InfoData/State
//   PLC/PLC Instance <-> EtherCAT Master EJxxxx/Beckhoff EJ7xxx/A_0029(EJ7211-9415-0031)
//     PlcTask Inputs/GVL_iXlinker.EtherCAT_Master_EJxxxx.Beckhoff_EJ7xxx.A_0029_EJ7211_9415_0031.DS402_Statusword.Statusword <-> DS402 Statusword/Statusword
//     PlcTask Inputs/GVL_iXlinker.EtherCAT_Master_EJxxxx.Beckhoff_EJ7xxx.A_0029_EJ7211_9415_0031.DS402_Position_actual_value.Position_actual_value <-> DS402 Position actual value/Position actual value
//     PlcTask Outputs/GVL_iXlinker.EtherCAT_Master_EJxxxx.Beckhoff_EJ7xxx.A_0029_EJ7211_9415_0031.DS402_Controlword.Controlword <-> DS402 Controlword/Controlword
//     PlcTask Outputs/GVL_iXlinker.EtherCAT_Master_EJxxxx.Beckhoff_EJ7xxx.A_0029_EJ7211_9415_0031.DS402_Target_velocity.Target_velocity <-> DS402 Target velocity/Target velocity
//     PlcTask Inputs/GVL_iXlinker.EtherCAT_Master_EJxxxx.Beckhoff_EJ7xxx.A_0029_EJ7211_9415_0031.WcState.WcState <-> WcState/WcState
//     PlcTask Inputs/GVL_iXlinker.EtherCAT_Master_EJxxxx.Beckhoff_EJ7xxx.A_0029_EJ7211_9415_0031.WcState.InputToggle <-> WcState/InputToggle
//     PlcTask Inputs/GVL_iXlinker.EtherCAT_Master_EJxxxx.Beckhoff_EJ7xxx.A_0029_EJ7211_9415_0031.InfoData.AdsAddr <-> InfoData/AdsAddr
//     PlcTask Inputs/GVL_iXlinker.EtherCAT_Master_EJxxxx.Beckhoff_EJ7xxx.A_0029_EJ7211_9415_0031.InfoData.DcOutputShift <-> InfoData/DcOutputShift
//     PlcTask Inputs/GVL_iXlinker.EtherCAT_Master_EJxxxx.Beckhoff_EJ7xxx.A_0029_EJ7211_9415_0031.InfoData.DcInputShift <-> InfoData/DcInputShift
//     PlcTask Inputs/GVL_iXlinker.EtherCAT_Master_EJxxxx.Beckhoff_EJ7xxx.A_0029_EJ7211_9415_0031.InfoData.Chn0 <-> InfoData/Chn0
//     PlcTask Inputs/GVL_iXlinker.EtherCAT_Master_EJxxxx.Beckhoff_EJ7xxx.A_0029_EJ7211_9415_0031.InfoData.State <-> InfoData/State
//   PLC/PLC Instance <-> EtherCAT Master EJxxxx/Beckhoff EJ7xxx/A_0030(EJ7211-9415-0032)
//     PlcTask Inputs/GVL_iXlinker.EtherCAT_Master_EJxxxx.Beckhoff_EJ7xxx.A_0030_EJ7211_9415_0032.DS402_Statusword.Statusword <-> DS402 Statusword/Statusword
//     PlcTask Inputs/GVL_iXlinker.EtherCAT_Master_EJxxxx.Beckhoff_EJ7xxx.A_0030_EJ7211_9415_0032.DS402_Position_actual_value.Position_actual_value <-> DS402 Position actual value/Position actual value
//     PlcTask Outputs/GVL_iXlinker.EtherCAT_Master_EJxxxx.Beckhoff_EJ7xxx.A_0030_EJ7211_9415_0032.DS402_Controlword.Controlword <-> DS402 Controlword/Controlword
//     PlcTask Outputs/GVL_iXlinker.EtherCAT_Master_EJxxxx.Beckhoff_EJ7xxx.A_0030_EJ7211_9415_0032.DS402_Target_velocity.Target_velocity <-> DS402 Target velocity/Target velocity
//     PlcTask Inputs/GVL_iXlinker.EtherCAT_Master_EJxxxx.Beckhoff_EJ7xxx.A_0030_EJ7211_9415_0032.WcState.WcState <-> WcState/WcState
//     PlcTask Inputs/GVL_iXlinker.EtherCAT_Master_EJxxxx.Beckhoff_EJ7xxx.A_0030_EJ7211_9415_0032.WcState.InputToggle <-> WcState/InputToggle
//     PlcTask Inputs/GVL_iXlinker.EtherCAT_Master_EJxxxx.Beckhoff_EJ7xxx.A_0030_EJ7211_9415_0032.InfoData.AdsAddr <-> InfoData/AdsAddr
//     PlcTask Inputs/GVL_iXlinker.EtherCAT_Master_EJxxxx.Beckhoff_EJ7xxx.A_0030_EJ7211_9415_0032.InfoData.DcOutputShift <-> InfoData/DcOutputShift
//     PlcTask Inputs/GVL_iXlinker.EtherCAT_Master_EJxxxx.Beckhoff_EJ7xxx.A_0030_EJ7211_9415_0032.InfoData.DcInputShift <-> InfoData/DcInputShift
//     PlcTask Inputs/GVL_iXlinker.EtherCAT_Master_EJxxxx.Beckhoff_EJ7xxx.A_0030_EJ7211_9415_0032.InfoData.Chn0 <-> InfoData/Chn0
//     PlcTask Inputs/GVL_iXlinker.EtherCAT_Master_EJxxxx.Beckhoff_EJ7xxx.A_0030_EJ7211_9415_0032.InfoData.State <-> InfoData/State
//   PLC/PLC Instance <-> EtherCAT Master EJxxxx/Beckhoff EJ7xxx/A_0031(EJ7334-0008-0016)
//     PlcTask Inputs/GVL_iXlinker.EtherCAT_Master_EJxxxx.Beckhoff_EJ7xxx.A_0031_EJ7334_0008_0016.DCM_Status_Channel_1.Status/Ready_to_enable <-> DCM Status Channel 1/Status/Ready to enable
//     PlcTask Inputs/GVL_iXlinker.EtherCAT_Master_EJxxxx.Beckhoff_EJ7xxx.A_0031_EJ7334_0008_0016.DCM_Status_Channel_2.Status/Ready_to_enable <-> DCM Status Channel 2/Status/Ready to enable
//     PlcTask Inputs/GVL_iXlinker.EtherCAT_Master_EJxxxx.Beckhoff_EJ7xxx.A_0031_EJ7334_0008_0016.DCM_Status_Channel_3.Status/Ready_to_enable <-> DCM Status Channel 3/Status/Ready to enable
//     PlcTask Inputs/GVL_iXlinker.EtherCAT_Master_EJxxxx.Beckhoff_EJ7xxx.A_0031_EJ7334_0008_0016.DCM_Status_Channel_4.Status/Ready_to_enable <-> DCM Status Channel 4/Status/Ready to enable
//     PlcTask Inputs/GVL_iXlinker.EtherCAT_Master_EJxxxx.Beckhoff_EJ7xxx.A_0031_EJ7334_0008_0016.DCM_Status_Channel_1.Status/Ready <-> DCM Status Channel 1/Status/Ready
//     PlcTask Inputs/GVL_iXlinker.EtherCAT_Master_EJxxxx.Beckhoff_EJ7xxx.A_0031_EJ7334_0008_0016.DCM_Status_Channel_2.Status/Ready <-> DCM Status Channel 2/Status/Ready
//     PlcTask Inputs/GVL_iXlinker.EtherCAT_Master_EJxxxx.Beckhoff_EJ7xxx.A_0031_EJ7334_0008_0016.DCM_Status_Channel_3.Status/Ready <-> DCM Status Channel 3/Status/Ready
//     PlcTask Inputs/GVL_iXlinker.EtherCAT_Master_EJxxxx.Beckhoff_EJ7xxx.A_0031_EJ7334_0008_0016.DCM_Status_Channel_4.Status/Ready <-> DCM Status Channel 4/Status/Ready
//     PlcTask Inputs/GVL_iXlinker.EtherCAT_Master_EJxxxx.Beckhoff_EJ7xxx.A_0031_EJ7334_0008_0016.DCM_Status_Channel_1.Status/Warning <-> DCM Status Channel 1/Status/Warning
//     PlcTask Inputs/GVL_iXlinker.EtherCAT_Master_EJxxxx.Beckhoff_EJ7xxx.A_0031_EJ7334_0008_0016.DCM_Status_Channel_2.Status/Warning <-> DCM Status Channel 2/Status/Warning
//     PlcTask Inputs/GVL_iXlinker.EtherCAT_Master_EJxxxx.Beckhoff_EJ7xxx.A_0031_EJ7334_0008_0016.DCM_Status_Channel_3.Status/Warning <-> DCM Status Channel 3/Status/Warning
//     PlcTask Inputs/GVL_iXlinker.EtherCAT_Master_EJxxxx.Beckhoff_EJ7xxx.A_0031_EJ7334_0008_0016.DCM_Status_Channel_4.Status/Warning <-> DCM Status Channel 4/Status/Warning
//     PlcTask Inputs/GVL_iXlinker.EtherCAT_Master_EJxxxx.Beckhoff_EJ7xxx.A_0031_EJ7334_0008_0016.DCM_Status_Channel_1.Status/Error <-> DCM Status Channel 1/Status/Error
//     PlcTask Inputs/GVL_iXlinker.EtherCAT_Master_EJxxxx.Beckhoff_EJ7xxx.A_0031_EJ7334_0008_0016.DCM_Status_Channel_2.Status/Error <-> DCM Status Channel 2/Status/Error
//     PlcTask Inputs/GVL_iXlinker.EtherCAT_Master_EJxxxx.Beckhoff_EJ7xxx.A_0031_EJ7334_0008_0016.DCM_Status_Channel_3.Status/Error <-> DCM Status Channel 3/Status/Error
//     PlcTask Inputs/GVL_iXlinker.EtherCAT_Master_EJxxxx.Beckhoff_EJ7xxx.A_0031_EJ7334_0008_0016.DCM_Status_Channel_4.Status/Error <-> DCM Status Channel 4/Status/Error
//     PlcTask Inputs/GVL_iXlinker.EtherCAT_Master_EJxxxx.Beckhoff_EJ7xxx.A_0031_EJ7334_0008_0016.DCM_Status_Channel_1.Status/Moving_positive <-> DCM Status Channel 1/Status/Moving positive
//     PlcTask Inputs/GVL_iXlinker.EtherCAT_Master_EJxxxx.Beckhoff_EJ7xxx.A_0031_EJ7334_0008_0016.DCM_Status_Channel_2.Status/Moving_positive <-> DCM Status Channel 2/Status/Moving positive
//     PlcTask Inputs/GVL_iXlinker.EtherCAT_Master_EJxxxx.Beckhoff_EJ7xxx.A_0031_EJ7334_0008_0016.DCM_Status_Channel_3.Status/Moving_positive <-> DCM Status Channel 3/Status/Moving positive
//     PlcTask Inputs/GVL_iXlinker.EtherCAT_Master_EJxxxx.Beckhoff_EJ7xxx.A_0031_EJ7334_0008_0016.DCM_Status_Channel_4.Status/Moving_positive <-> DCM Status Channel 4/Status/Moving positive
//     PlcTask Inputs/GVL_iXlinker.EtherCAT_Master_EJxxxx.Beckhoff_EJ7xxx.A_0031_EJ7334_0008_0016.DCM_Status_Channel_1.Status/Moving_negative <-> DCM Status Channel 1/Status/Moving negative
//     PlcTask Inputs/GVL_iXlinker.EtherCAT_Master_EJxxxx.Beckhoff_EJ7xxx.A_0031_EJ7334_0008_0016.DCM_Status_Channel_2.Status/Moving_negative <-> DCM Status Channel 2/Status/Moving negative
//     PlcTask Inputs/GVL_iXlinker.EtherCAT_Master_EJxxxx.Beckhoff_EJ7xxx.A_0031_EJ7334_0008_0016.DCM_Status_Channel_3.Status/Moving_negative <-> DCM Status Channel 3/Status/Moving negative
//     PlcTask Inputs/GVL_iXlinker.EtherCAT_Master_EJxxxx.Beckhoff_EJ7xxx.A_0031_EJ7334_0008_0016.DCM_Status_Channel_4.Status/Moving_negative <-> DCM Status Channel 4/Status/Moving negative
//     PlcTask Inputs/GVL_iXlinker.EtherCAT_Master_EJxxxx.Beckhoff_EJ7xxx.A_0031_EJ7334_0008_0016.DCM_Status_Channel_1.Status/Limit_x <-> DCM Status Channel 1/Status/Limit
//     PlcTask Inputs/GVL_iXlinker.EtherCAT_Master_EJxxxx.Beckhoff_EJ7xxx.A_0031_EJ7334_0008_0016.DCM_Status_Channel_2.Status/Limit_x <-> DCM Status Channel 2/Status/Limit
//     PlcTask Inputs/GVL_iXlinker.EtherCAT_Master_EJxxxx.Beckhoff_EJ7xxx.A_0031_EJ7334_0008_0016.DCM_Status_Channel_3.Status/Limit_x <-> DCM Status Channel 3/Status/Limit
//     PlcTask Inputs/GVL_iXlinker.EtherCAT_Master_EJxxxx.Beckhoff_EJ7xxx.A_0031_EJ7334_0008_0016.DCM_Status_Channel_4.Status/Limit_x <-> DCM Status Channel 4/Status/Limit
//     PlcTask Inputs/GVL_iXlinker.EtherCAT_Master_EJxxxx.Beckhoff_EJ7xxx.A_0031_EJ7334_0008_0016.DCM_Status_Channel_1.Status/TxPDO_Toggle <-> DCM Status Channel 1/Status/TxPDO Toggle
//     PlcTask Inputs/GVL_iXlinker.EtherCAT_Master_EJxxxx.Beckhoff_EJ7xxx.A_0031_EJ7334_0008_0016.DCM_Status_Channel_2.Status/TxPDO_Toggle <-> DCM Status Channel 2/Status/TxPDO Toggle
//     PlcTask Inputs/GVL_iXlinker.EtherCAT_Master_EJxxxx.Beckhoff_EJ7xxx.A_0031_EJ7334_0008_0016.DCM_Status_Channel_3.Status/TxPDO_Toggle <-> DCM Status Channel 3/Status/TxPDO Toggle
//     PlcTask Inputs/GVL_iXlinker.EtherCAT_Master_EJxxxx.Beckhoff_EJ7xxx.A_0031_EJ7334_0008_0016.DCM_Status_Channel_4.Status/TxPDO_Toggle <-> DCM Status Channel 4/Status/TxPDO Toggle
//     PlcTask Outputs/GVL_iXlinker.EtherCAT_Master_EJxxxx.Beckhoff_EJ7xxx.A_0031_EJ7334_0008_0016.DCM_Outputs_Channel_1.Control/Enable <-> DCM Outputs Channel 1/Control/Enable
//     PlcTask Outputs/GVL_iXlinker.EtherCAT_Master_EJxxxx.Beckhoff_EJ7xxx.A_0031_EJ7334_0008_0016.DCM_Outputs_Channel_2.Control/Enable <-> DCM Outputs Channel 2/Control/Enable
//     PlcTask Outputs/GVL_iXlinker.EtherCAT_Master_EJxxxx.Beckhoff_EJ7xxx.A_0031_EJ7334_0008_0016.DCM_Outputs_Channel_3.Control/Enable <-> DCM Outputs Channel 3/Control/Enable
//     PlcTask Outputs/GVL_iXlinker.EtherCAT_Master_EJxxxx.Beckhoff_EJ7xxx.A_0031_EJ7334_0008_0016.DCM_Outputs_Channel_4.Control/Enable <-> DCM Outputs Channel 4/Control/Enable
//     PlcTask Outputs/GVL_iXlinker.EtherCAT_Master_EJxxxx.Beckhoff_EJ7xxx.A_0031_EJ7334_0008_0016.DCM_Outputs_Channel_1.Control/Reset <-> DCM Outputs Channel 1/Control/Reset
//     PlcTask Outputs/GVL_iXlinker.EtherCAT_Master_EJxxxx.Beckhoff_EJ7xxx.A_0031_EJ7334_0008_0016.DCM_Outputs_Channel_2.Control/Reset <-> DCM Outputs Channel 2/Control/Reset
//     PlcTask Outputs/GVL_iXlinker.EtherCAT_Master_EJxxxx.Beckhoff_EJ7xxx.A_0031_EJ7334_0008_0016.DCM_Outputs_Channel_3.Control/Reset <-> DCM Outputs Channel 3/Control/Reset
//     PlcTask Outputs/GVL_iXlinker.EtherCAT_Master_EJxxxx.Beckhoff_EJ7xxx.A_0031_EJ7334_0008_0016.DCM_Outputs_Channel_4.Control/Reset <-> DCM Outputs Channel 4/Control/Reset
//     PlcTask Outputs/GVL_iXlinker.EtherCAT_Master_EJxxxx.Beckhoff_EJ7xxx.A_0031_EJ7334_0008_0016.DCM_Outputs_Channel_1.Velocity <-> DCM Outputs Channel 1/Velocity
//     PlcTask Outputs/GVL_iXlinker.EtherCAT_Master_EJxxxx.Beckhoff_EJ7xxx.A_0031_EJ7334_0008_0016.DCM_Outputs_Channel_2.Velocity <-> DCM Outputs Channel 2/Velocity
//     PlcTask Outputs/GVL_iXlinker.EtherCAT_Master_EJxxxx.Beckhoff_EJ7xxx.A_0031_EJ7334_0008_0016.DCM_Outputs_Channel_3.Velocity <-> DCM Outputs Channel 3/Velocity
//     PlcTask Outputs/GVL_iXlinker.EtherCAT_Master_EJxxxx.Beckhoff_EJ7xxx.A_0031_EJ7334_0008_0016.DCM_Outputs_Channel_4.Velocity <-> DCM Outputs Channel 4/Velocity
//     PlcTask Inputs/GVL_iXlinker.EtherCAT_Master_EJxxxx.Beckhoff_EJ7xxx.A_0031_EJ7334_0008_0016.WcState.WcState <-> WcState/WcState
//     PlcTask Inputs/GVL_iXlinker.EtherCAT_Master_EJxxxx.Beckhoff_EJ7xxx.A_0031_EJ7334_0008_0016.WcState.InputToggle <-> WcState/InputToggle
//     PlcTask Inputs/GVL_iXlinker.EtherCAT_Master_EJxxxx.Beckhoff_EJ7xxx.A_0031_EJ7334_0008_0016.InfoData.AdsAddr <-> InfoData/AdsAddr
//     PlcTask Inputs/GVL_iXlinker.EtherCAT_Master_EJxxxx.Beckhoff_EJ7xxx.A_0031_EJ7334_0008_0016.InfoData.State <-> InfoData/State
//   PLC/PLC Instance <-> EtherCAT Master EJxxxx/Beckhoff EJ7xxx/A_0032(EJ7411-0000-0018)
//     PlcTask Inputs/GVL_iXlinker.EtherCAT_Master_EJxxxx.Beckhoff_EJ7xxx.A_0032_EJ7411_0000_0018.FB_Position.Position <-> FB Position/Position
//     PlcTask Inputs/GVL_iXlinker.EtherCAT_Master_EJxxxx.Beckhoff_EJ7xxx.A_0032_EJ7411_0000_0018.DRV_Statusword.Statusword <-> DRV Statusword/Statusword
//     PlcTask Inputs/GVL_iXlinker.EtherCAT_Master_EJxxxx.Beckhoff_EJ7xxx.A_0032_EJ7411_0000_0018.DRV_Following_error_actual_value.Following_error_actual_value <-> DRV Following error actual value/Following error actual value
//     PlcTask Outputs/GVL_iXlinker.EtherCAT_Master_EJxxxx.Beckhoff_EJ7xxx.A_0032_EJ7411_0000_0018.DRV_Controlword.Controlword <-> DRV Controlword/Controlword
//     PlcTask Outputs/GVL_iXlinker.EtherCAT_Master_EJxxxx.Beckhoff_EJ7xxx.A_0032_EJ7411_0000_0018.DRV_Target_position.Target_position <-> DRV Target position/Target position
//     PlcTask Inputs/GVL_iXlinker.EtherCAT_Master_EJxxxx.Beckhoff_EJ7xxx.A_0032_EJ7411_0000_0018.WcState.WcState <-> WcState/WcState
//     PlcTask Inputs/GVL_iXlinker.EtherCAT_Master_EJxxxx.Beckhoff_EJ7xxx.A_0032_EJ7411_0000_0018.WcState.InputToggle <-> WcState/InputToggle
//     PlcTask Inputs/GVL_iXlinker.EtherCAT_Master_EJxxxx.Beckhoff_EJ7xxx.A_0032_EJ7411_0000_0018.InfoData.AdsAddr <-> InfoData/AdsAddr
//     PlcTask Inputs/GVL_iXlinker.EtherCAT_Master_EJxxxx.Beckhoff_EJ7xxx.A_0032_EJ7411_0000_0018.InfoData.DcOutputShift <-> InfoData/DcOutputShift
//     PlcTask Inputs/GVL_iXlinker.EtherCAT_Master_EJxxxx.Beckhoff_EJ7xxx.A_0032_EJ7411_0000_0018.InfoData.DcInputShift <-> InfoData/DcInputShift
//     PlcTask Inputs/GVL_iXlinker.EtherCAT_Master_EJxxxx.Beckhoff_EJ7xxx.A_0032_EJ7411_0000_0018.InfoData.Chn0 <-> InfoData/Chn0
//     PlcTask Inputs/GVL_iXlinker.EtherCAT_Master_EJxxxx.Beckhoff_EJ7xxx.A_0032_EJ7411_0000_0018.InfoData.Chn1 <-> InfoData/Chn1
//     PlcTask Inputs/GVL_iXlinker.EtherCAT_Master_EJxxxx.Beckhoff_EJ7xxx.A_0032_EJ7411_0000_0018.InfoData.State <-> InfoData/State
//   PLC/PLC Instance <-> EtherCAT Master EJxxxx/Beckhoff EJ9xxx
//     PlcTask Inputs/GVL_iXlinker.EtherCAT_Master_EJxxxx.Beckhoff_EJ9xxx.InfoData.State <-> InfoData/State
//   PLC/PLC Instance <-> EtherCAT Master EJxxxx/Beckhoff EJ9xxx/Beckhoff EJ9xxxEK1122
//     PlcTask Inputs/GVL_iXlinker.EtherCAT_Master_EJxxxx.Beckhoff_EJ9xxx.Beckhoff_EJ9xxxEK1122.InfoData.State <-> InfoData/State
//   PLC/PLC Instance <-> EtherCAT Master EJxxxx/Beckhoff EJ9xxx/Beckhoff EJ9xxxEK1122/Beckhoff EJ9xxxsub EK1100
//     PlcTask Inputs/GVL_iXlinker.EtherCAT_Master_EJxxxx.Beckhoff_EJ9xxx.Beckhoff_EJ9xxxEK1122.Beckhoff_EJ9xxxsub_EK1100.InfoData.State <-> InfoData/State
//   PLC/PLC Instance <-> EtherCAT Master EJxxxx/Beckhoff EJ9xxx/A_0001(EJ9001-0000-0016)
//     PlcTask Inputs/GVL_iXlinker.EtherCAT_Master_EJxxxx.Beckhoff_EJ9xxx.A_0001_EJ9001_0000_0016.InfoData.State <-> InfoData/State
//   PLC/PLC Instance <-> EtherCAT Master EJxxxx/Beckhoff EJ9xxx/A_0002(EJ9505-0000-0016)
//     PlcTask Inputs/GVL_iXlinker.EtherCAT_Master_EJxxxx.Beckhoff_EJ9xxx.A_0002_EJ9505_0000_0016.Status_Uo.Power_OK <-> Status Uo/Power OK
//     PlcTask Inputs/GVL_iXlinker.EtherCAT_Master_EJxxxx.Beckhoff_EJ9xxx.A_0002_EJ9505_0000_0016.Status_Uo.Overload <-> Status Uo/Overload
//     PlcTask Inputs/GVL_iXlinker.EtherCAT_Master_EJxxxx.Beckhoff_EJ9xxx.A_0002_EJ9505_0000_0016.WcState.WcState <-> WcState/WcState
//     PlcTask Inputs/GVL_iXlinker.EtherCAT_Master_EJxxxx.Beckhoff_EJ9xxx.A_0002_EJ9505_0000_0016.WcState.InputToggle <-> WcState/InputToggle
//     PlcTask Inputs/GVL_iXlinker.EtherCAT_Master_EJxxxx.Beckhoff_EJ9xxx.A_0002_EJ9505_0000_0016.InfoData.State <-> InfoData/State
//   PLC/PLC Instance <-> EtherCAT Master EJxxxx/Beckhoff EJ9xxx/A_0003(EJ9576-0000-0018)
//     PlcTask Inputs/GVL_iXlinker.EtherCAT_Master_EJxxxx.Beckhoff_EJ9xxx.A_0003_EJ9576_0000_0018.BCT_Inputs.Terminal_Overtemperature <-> BCT Inputs/Terminal Overtemperature
//     PlcTask Inputs/GVL_iXlinker.EtherCAT_Master_EJxxxx.Beckhoff_EJ9xxx.A_0003_EJ9576_0000_0018.BCT_Inputs.I2T_error <-> BCT Inputs/I2T error
//     PlcTask Inputs/GVL_iXlinker.EtherCAT_Master_EJxxxx.Beckhoff_EJ9xxx.A_0003_EJ9576_0000_0018.BCT_Inputs.I2T_warning <-> BCT Inputs/I2T warning
//     PlcTask Inputs/GVL_iXlinker.EtherCAT_Master_EJxxxx.Beckhoff_EJ9xxx.A_0003_EJ9576_0000_0018.BCT_Inputs.Overvoltage <-> BCT Inputs/Overvoltage
//     PlcTask Inputs/GVL_iXlinker.EtherCAT_Master_EJxxxx.Beckhoff_EJ9xxx.A_0003_EJ9576_0000_0018.BCT_Inputs.Undervoltage <-> BCT Inputs/Undervoltage
//     PlcTask Inputs/GVL_iXlinker.EtherCAT_Master_EJxxxx.Beckhoff_EJ9xxx.A_0003_EJ9576_0000_0018.BCT_Inputs.Chopper_on <-> BCT Inputs/Chopper on
//     PlcTask Inputs/GVL_iXlinker.EtherCAT_Master_EJxxxx.Beckhoff_EJ9xxx.A_0003_EJ9576_0000_0018.BCT_Inputs.Input_cycle_counter <-> BCT Inputs/Input cycle counter
//     PlcTask Inputs/GVL_iXlinker.EtherCAT_Master_EJxxxx.Beckhoff_EJ9xxx.A_0003_EJ9576_0000_0018.BCT_Inputs.DC_link_voltage <-> BCT Inputs/DC link voltage
//     PlcTask Inputs/GVL_iXlinker.EtherCAT_Master_EJxxxx.Beckhoff_EJ9xxx.A_0003_EJ9576_0000_0018.BCT_Inputs.Resistor_current <-> BCT Inputs/Resistor current
//     PlcTask Inputs/GVL_iXlinker.EtherCAT_Master_EJxxxx.Beckhoff_EJ9xxx.A_0003_EJ9576_0000_0018.BCT_Inputs.Duty_cylce <-> BCT Inputs/Duty cylce
